// TIA Portal project "03PLC" (V15)

(* hardware
DEVICE "S7-1200 station_1"  S7-1200 Station
   slot 0: "Rack_0"  S7-1200 Rack  Rack  V1.0
   slot 1: "PLC_1"  CPU 1215C DC/DC/DC  6ES7 215-1AG40-0XB0  V4.0
   slot 2: "DI 16x24VDC/DQ 16xRelay_1"  SM 1223 DI16/DQ16 x relay  6ES7 223-1PL32-0XB0  V2.0
   slot 3: "DI 16x24VDC/DQ 16xRelay_2"  SM 1223 DI16/DQ16 x relay  6ES7 223-1PL32-0XB0  V2.0
   slot 4: "DI 16x24VDC_1"  6ES7 221-1BH32-0XB0  V2.0
   slot 5: "DI 16x24VDC_2"  6ES7 221-1BH32-0XB0  V2.0
DEVICE "HMI_1"  TP700 Comfort
   slot 0: "HMI_1"  TP700 Comfort  6AV2 124-0GC01-0AX0  15.0.0.0
   slot 1: "HMI_RT_1"  TP700 Comfort  6AV2 124-0GC01-0AX0  15.0.0.0
   slot 5: "HMI_1.IE_CP_1"  PROFINET Interface  15.0.0.0
      slot 1: "PROFINET Interface_1"  PROFINET Interface
         slot 1: "Port_1"  Port
         slot 2: "Port_2"  Port
   slot 7: "HMI_1.MPI/DP_CP_1"  MPI/DP Interface  15.0.0.0
DEVICE "GSD device_1"  GSD.Device.PN
   slot 0: "机架"  Rack  V1.0
   slot 0: "RFID"  RF180C V2.2  6GT2 002-0JD00  2.0
      slot 0: "Standard"  Standard
      slot 1: "RF180C Interface"  RF180C Interface
         slot 1: "Port 1"  Port 1
         slot 2: "Port 2"  Port 2
      slot 1: "2x RS422 channels RFID_1"  2x RS422 channels RFID
         slot 0: "2x RS422 channels RFID"  2x RS422 channels RFID
*)

// ===== PLC "PLC_1"  CPU 1215C DC/DC/DC =====

VAR_GLOBAL   // PLC tag table "默认变量表"
   "System_Byte" AT %MB1 : Byte;
   "FirstScan" AT %M1.0 : Bool;
   "DiagStatusUpdate" AT %M1.1 : Bool;
   "AlwaysTRUE" AT %M1.2 : Bool;
   "AlwaysFALSE" AT %M1.3 : Bool;
   "Clock_Byte" AT %MB0 : Byte;
   "Clock_10Hz" AT %M0.0 : Bool;
   "Clock_5Hz" AT %M0.1 : Bool;
   "Clock_2.5Hz" AT %M0.2 : Bool;
   "Clock_2Hz" AT %M0.3 : Bool;
   "Clock_1.25Hz" AT %M0.4 : Bool;
   "Clock_1Hz" AT %M0.5 : Bool;
   "Clock_0.625Hz" AT %M0.6 : Bool;
   "Clock_0.5Hz" AT %M0.7 : Bool;
   "Tag_1" AT %M9.0 : Bool;
   "Tag_2" AT %MW10 : Word;
   "Tag_69" AT %M100.0 : Bool;
   "Tag_70" AT %M200.0 : Bool;
   "Tag_71" AT %I0.2 : Bool;
   "Tag_72" AT %Q5.0 : Bool;
END_VAR

VAR_GLOBAL   // PLC tag table "变量表_1"
   "Tag_3" AT %I2.0 : Bool;
   "Tag_4" AT %I2.1 : Bool;
   "Tag_5" AT %I2.2 : Bool;
   "Tag_6" AT %I2.3 : Bool;
   "Tag_7" AT %I2.4 : Bool;
   "Tag_8" AT %I2.5 : Bool;
   "Tag_9" AT %I2.6 : Bool;
   "Tag_10" AT %I2.7 : Bool;
   "Tag_11" AT %Q2.0 : Bool;
   "Tag_12" AT %Q2.1 : Bool;
   "Tag_13" AT %Q2.2 : Bool;
   "Tag_14" AT %Q2.3 : Bool;
   "Tag_15" AT %Q2.4 : Bool;
   "Tag_16" AT %Q2.5 : Bool;
   "Tag_17" AT %Q2.6 : Bool;
   "Tag_18" AT %Q2.7 : Bool;
   "Tag_19" AT %I3.0 : Bool;
   "Tag_20" AT %I5.0 : Bool;
   "Tag_21" AT %I5.2 : Bool;
   "Tag_22" AT %Q0.4 : Bool;
   "Tag_23" AT %Q0.5 : Bool;
END_VAR

VAR_GLOBAL   // PLC tag table "变量表_2"
   "Tag_24" AT %I4.0 : Bool;
   "Tag_25" AT %I4.1 : Bool;
   "Tag_26" AT %I4.2 : Bool;
   "Tag_27" AT %I4.3 : Bool;
   "Tag_28" AT %I4.4 : Bool;
   "Tag_29" AT %I4.5 : Bool;
   "Tag_30" AT %I4.6 : Bool;
   "Tag_31" AT %Q4.0 : Bool;
   "Tag_32" AT %Q4.1 : Bool;
   "Tag_33" AT %Q4.2 : Bool;
   "Tag_34" AT %Q4.3 : Bool;
   "Tag_35" AT %Q4.4 : Bool;
   "Tag_36" AT %Q4.5 : Bool;
   "Tag_37" AT %Q4.6 : Bool;
   "Tag_38" AT %Q4.7 : Bool;
END_VAR

VAR_GLOBAL   // PLC tag table "变量表_3"
   "Tag_39" AT %I6.0 : Bool;
   "Tag_40" AT %I6.1 : Bool;
   "Tag_41" AT %I6.2 : Bool;
   "Tag_42" AT %I6.3 : Bool;
   "Tag_43" AT %I6.4 : Bool;
   "Tag_44" AT %I6.5 : Bool;
   "Tag_45" AT %I6.6 : Bool;
   "Tag_46" AT %I6.7 : Bool;
   "Tag_47" AT %I7.0 : Bool;
   "Tag_48" AT %I7.1 : Bool;
   "Tag_49" AT %I7.2 : Bool;
   "Tag_50" AT %I7.3 : Bool;
   "Tag_51" AT %I7.4 : Bool;
   "Tag_52" AT %I7.5 : Bool;
   "Tag_53" AT %I7.6 : Bool;
   "Tag_54" AT %I8.0 : Bool;
   "Tag_55" AT %I8.1 : Bool;
   "Tag_56" AT %I8.2 : Bool;
   "Tag_57" AT %I8.3 : Bool;
   "Tag_58" AT %I8.4 : Bool;
   "Tag_59" AT %I8.5 : Bool;
   "Tag_60" AT %I8.6 : Bool;
   "Tag_61" AT %I8.7 : Bool;
   "Tag_62" AT %I9.0 : Bool;
   "Tag_63" AT %I9.1 : Bool;
   "Tag_64" AT %I9.2 : Bool;
   "Tag_65" AT %I9.3 : Bool;
   "Tag_66" AT %I9.4 : Bool;
   "Tag_67" AT %I9.5 : Bool;
   "Tag_68" AT %I9.6 : Bool;
END_VAR

TYPE "用户数据类型_1"
   STRUCT
      场次 : Int;
      种类 : Int;
      材质 : Int;
      状态 : Int;
   END_STRUCT;
END_TYPE

DATA_BLOCK "mes数据块"   // DB1
{ S7_Optimized_Access := 'FALSE' }
VERSION : 0.1
   VAR
      mes给plc : Struct
         mes命令 : Struct
            "1" : Int;
            "2" : Int;
            "3" : Int;
            "4" : Int;
            "5" : Int;
            "6" : Int;
            "7" : Int;
            "8" : Int;
            "9" : Int;
            "10" : Int;
         END_STRUCT;
         mes反馈车床 : Struct
            "1" : Int;
            "2" : Int;
            "3" : Int;
            "4" : Int;
            "5" : Int;
         END_STRUCT;
         mes反馈cnc : Struct
            "1" : Int;
            "2" : Int;
            "3" : Int;
            "4" : Int;
            "5" : Int;
         END_STRUCT;
      END_STRUCT;
      plc给mes : Struct
         plc命令车床 : Struct
            "1" : Int;
            "2" : Int;
            "3" : Int;
            "4" : Int;
            "5" : Int;
         END_STRUCT;
         plc命令cnc : Struct
            "1" : Int;
            "2" : Int;
            "3" : Int;
            "4" : Int;
            "5" : Int;
         END_STRUCT;
         plc反馈 : Struct
            "1" : Int;
            "2" : Int;
            "3" : Int;
            "4" : Int;
            "5" : Int;
            "6" : Int;
            "7" : Int;
            "8" : Int;
            "9" : Int;
            "10" : Int;
         END_STRUCT;
         机器人状态 : Struct
            "1" : Int;
            "2" : Int;
            "3" : Int;
            "4" : Int;
            "5" : Int;
            "6" : Int;
            "7" : Int;
            "8" : Int;
            "9" : Int;
            "10" : Int;
            "11" : Int;
         END_STRUCT;
         保留 : Array[0..8] of Word;
      END_STRUCT;
      仓库 : Struct
         "1" : Bool;
         "2" : Bool;
         "3" : Bool;
         "4" : Bool;
         "5" : Bool;
         "6" : Bool;
         "7" : Bool;
         "8" : Bool;
         "9" : Bool;
         "10" : Bool;
         "11" : Bool;
         "12" : Bool;
         "13" : Bool;
         "14" : Bool;
         "15" : Bool;
         保留 : Bool;
         "16" : Bool;
         "17" : Bool;
         "18" : Bool;
         "19" : Bool;
         "20" : Bool;
         "21" : Bool;
         "22" : Bool;
         "23" : Bool;
         "24" : Bool;
         "25" : Bool;
         "26" : Bool;
         "27" : Bool;
         "28" : Bool;
         "29" : Bool;
         "30" : Bool;
      END_STRUCT;
      保留 : Array[0..47] of Bool;
      机床状态 : Array[0..79] of Bool;
      工件 : Array[1..30] of "用户数据类型_1";
      测量 : Array[1..10] of Int;
   END_VAR
BEGIN
END_DATA_BLOCK

DATA_BLOCK "机器人数据块"   // DB2
{ S7_Optimized_Access := 'FALSE' }
VERSION : 0.1
   VAR
      plc给机器人 : Struct
         "1" : Int;
         "2" : Int;
         "3" : Int;
         "4" : Int;
         "5" : Int;
         "6" : Int;
         "7" : Int;
         "8" : Int;
         "9" : Int;
         "10" : Int;
         "11" : Int;
         "12" : Int;
         "13" : Int;
         "14" : Int;
         "15" : Int;
         "16" : Int;
      END_STRUCT;
      机器人给plc : Struct
         "1" : Int;
         "2" : Int;
         "3" : Int;
         "4" : Int;
         "5" : Int;
         "6" : Int;
         "7" : Int;
         "8" : Int;
         "9" : Int;
         "10" : Int;
         "11" : Int;
         "12" : Int;
         "13" : Int;
         "14" : Int;
         "15" : Int;
         "16" : Int;
      END_STRUCT;
      机器人状态 : Struct
         "1" : Real;
         "2" : Real;
         "3" : Real;
         "4" : Real;
         "5" : Real;
         "6" : Real;
         "7" : Real;
         "8" : Real;
         "9" : Real;
         "10" : Real;
         "11" : Real;
         "12" : Real;
         "13" : Real;
         "14" : Real;
         "15" : Real;
         "16" : Real;
      END_STRUCT;
   END_VAR
BEGIN
END_DATA_BLOCK

DATA_BLOCK "hmi"   // DB3
{ S7_Optimized_Access := 'TRUE' }
VERSION : 0.1
   VAR
      车床卡盘 : Bool;
      cnc卡盘 : Bool;
      零点夹具 : Bool;
      车床门开关 : Bool;
      铣床门开关 : Bool;
      机器人home位 : Bool;
      mes订单已下发 : Bool;
      自动 : Bool;
      手动 : Bool;
      清理 : Time;
      间隔 : Time;
      种类 : Int;
      状态 : Int;
      当前仓位 : Int;
   END_VAR
BEGIN
END_DATA_BLOCK

DATA_BLOCK "mes_DB"   // DB4
{ S7_Optimized_Access := 'TRUE' }
VERSION : 0.1
// stored: InstanceOfName mes
"mes"
BEGIN
END_DATA_BLOCK

DATA_BLOCK "rfid_DB"   // DB7
{ S7_Optimized_Access := 'TRUE' }
VERSION : 0.1
// stored: InstanceOfName rfid
"rfid"
BEGIN
END_DATA_BLOCK

DATA_BLOCK "车床_DB"   // DB8
{ S7_Optimized_Access := 'TRUE' }
VERSION : 0.1
// stored: InstanceOfName 车床
"车床"
BEGIN
END_DATA_BLOCK

DATA_BLOCK "铣床_DB"   // DB9
{ S7_Optimized_Access := 'TRUE' }
VERSION : 0.1
// stored: InstanceOfName 铣床
"铣床"
BEGIN
END_DATA_BLOCK

DATA_BLOCK "机器人通讯_DB"   // DB10
{ S7_Optimized_Access := 'TRUE' }
VERSION : 0.1
// stored: InstanceOfName 机器人通讯
"机器人通讯"
BEGIN
END_DATA_BLOCK

DATA_BLOCK "机床状态_DB"   // DB11
{ S7_Optimized_Access := 'TRUE' }
VERSION : 0.1
// stored: InstanceOfName 机床状态
"机床状态"
BEGIN
END_DATA_BLOCK

DATA_BLOCK "测量_DB"   // DB12
{ S7_Optimized_Access := 'TRUE' }
VERSION : 0.1
// stored: InstanceOfName 测量
"测量"
BEGIN
END_DATA_BLOCK

DATA_BLOCK "有无料_DB"   // DB13
{ S7_Optimized_Access := 'TRUE' }
VERSION : 0.1
// stored: InstanceOfName 有无料
"有无料"
BEGIN
END_DATA_BLOCK

// folder: rfid

DATA_BLOCK "connect"   // DB5
{ S7_Optimized_Access := 'TRUE' }
VERSION : 0.1
   VAR
      connect : IID_HW_CONNECT;
   END_VAR
BEGIN
END_DATA_BLOCK

DATA_BLOCK "读写"   // DB6
{ S7_Optimized_Access := 'FALSE' }
VERSION : 0.1
   VAR
      读 : Array[0..1024] of Byte;
      写 : Array[0..1024] of Byte;
   END_VAR
BEGIN
END_DATA_BLOCK

// folder: (top level)

FUNCTION_BLOCK "机器人通讯"   // FB1, LAD
{ S7_Optimized_Access := 'TRUE' }
VERSION : 0.1
   VAR
      MB_CLIENT_Instance : MB_CLIENT;
      w1 : Bool;
      w2 : Bool;
      w3 : Bool;
      m1 : Bool;
      m2 : Bool;
      m3 : Bool;
      c1 : Bool;
      c2 : Bool;
      c3 : Bool;
      s1 : Word;
      s2 : Word;
      s3 : Word;
      轴1 : Int;
      轴2 : Int;
      轴3 : Int;
      轴4 : Int;
      轴5 : Int;
      轴6 : Int;
      轴7 : Int;
   END_VAR
BEGIN

REGION Network 1
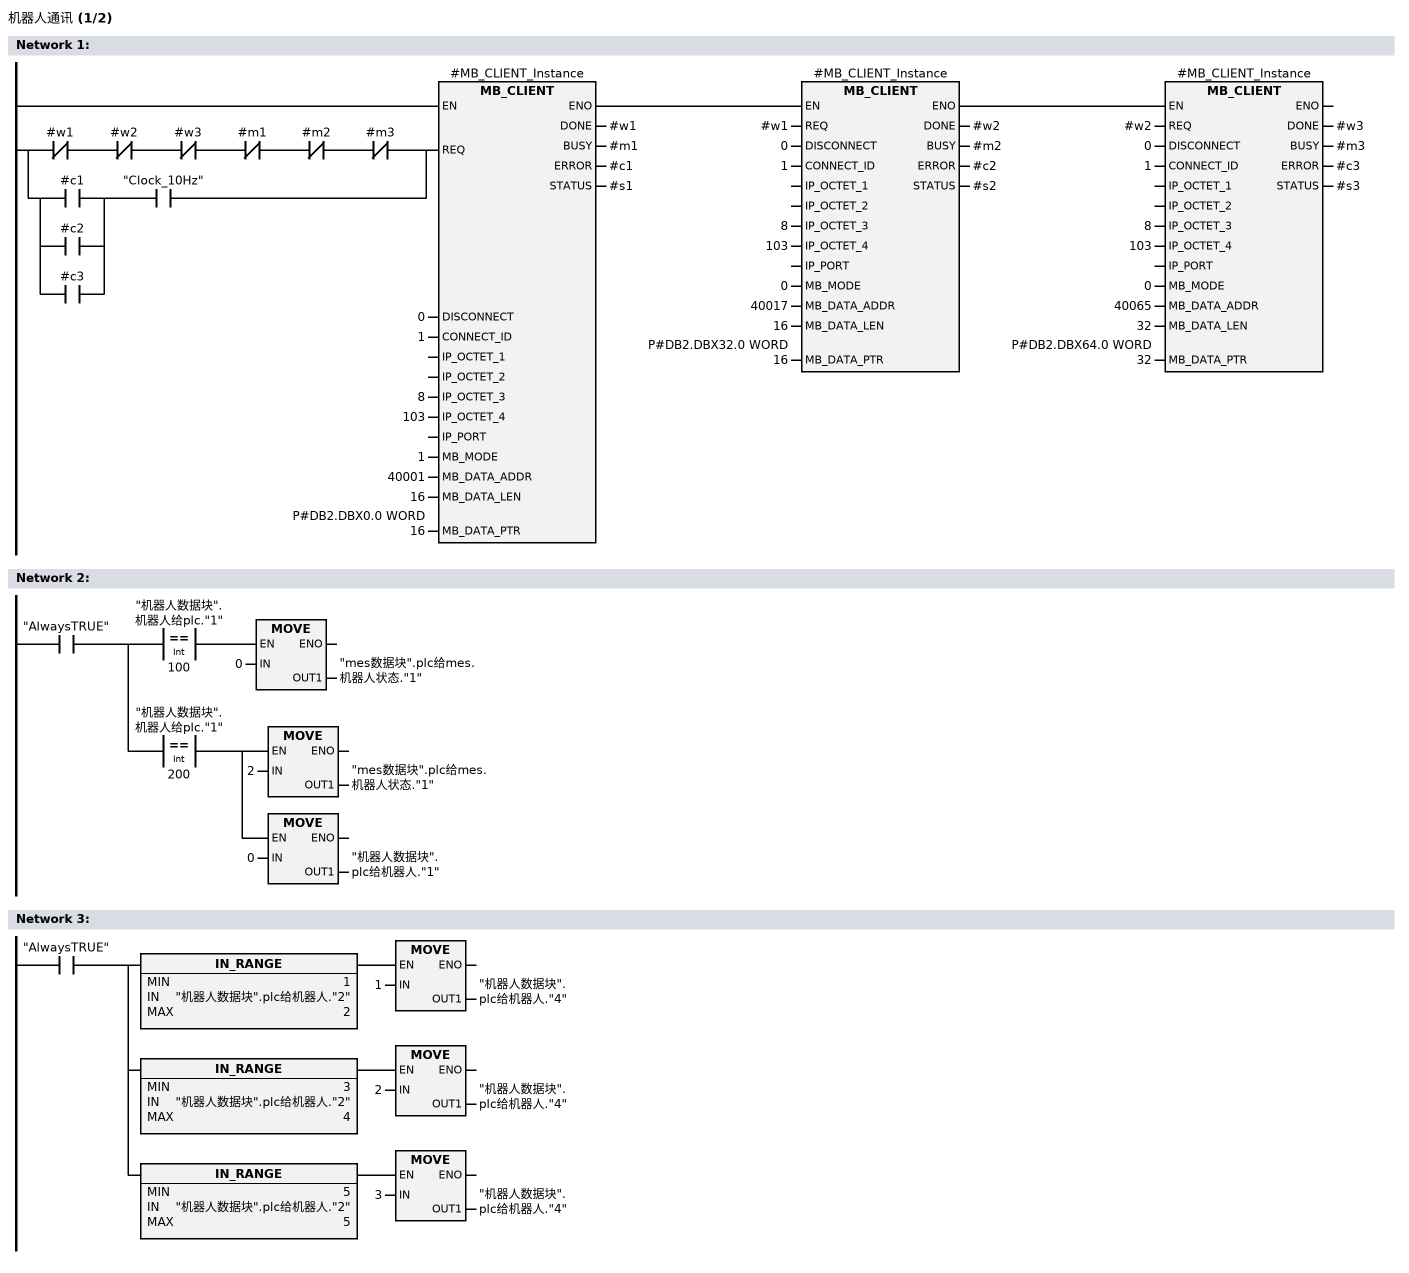
   // ENO of a box is taken as its EN; it also drops when the box reports an error
   #MB_CLIENT_Instance(REQ := (NOT #w1 AND NOT #w2 AND NOT #w3 AND NOT #m1 AND NOT #m2 AND NOT #m3) OR ((#c1 OR #c2 OR #c3) AND "Clock_10Hz"),   // MB_CLIENT
                       DISCONNECT := 0,
                       CONNECT_ID := 1,
                       IP_OCTET_3 := 8,
                       IP_OCTET_4 := 103,
                       MB_MODE := 1,
                       MB_DATA_ADDR := 40001,
                       MB_DATA_LEN := 16,
                       MB_DATA_PTR := P#DB2.DBX0.0 WORD 16,
                       DONE => #w1,
                       BUSY => #m1,
                       ERROR => #c1,
                       STATUS => #s1);
   #MB_CLIENT_Instance(REQ := #w1,   // MB_CLIENT
                       DISCONNECT := 0,
                       CONNECT_ID := 1,
                       IP_OCTET_3 := 8,
                       IP_OCTET_4 := 103,
                       MB_MODE := 0,
                       MB_DATA_ADDR := 40017,
                       MB_DATA_LEN := 16,
                       MB_DATA_PTR := P#DB2.DBX32.0 WORD 16,
                       DONE => #w2,
                       BUSY => #m2,
                       ERROR => #c2,
                       STATUS => #s2);
   #MB_CLIENT_Instance(REQ := #w2,   // MB_CLIENT
                       DISCONNECT := 0,
                       CONNECT_ID := 1,
                       IP_OCTET_3 := 8,
                       IP_OCTET_4 := 103,
                       MB_MODE := 0,
                       MB_DATA_ADDR := 40065,
                       MB_DATA_LEN := 32,
                       MB_DATA_PTR := P#DB2.DBX64.0 WORD 32,
                       DONE => #w3,
                       BUSY => #m3,
                       ERROR => #c3,
                       STATUS => #s3);
END_REGION

REGION Network 2
   RUNG wire#powerrail
      Contact( "AlwaysTRUE" )
      wire#w1
      { S7_Templates := "SrcType := Int" } EQ_Contact(in1 := "机器人数据块".机器人给plc."1", in2 := 100)
      Move(in := 0, out1 => "mes数据块".plc给mes.机器人状态."1")
   END_RUNG
   RUNG wire#w1
      { S7_Templates := "SrcType := Int" } EQ_Contact(in1 := "机器人数据块".机器人给plc."1", in2 := 200)
      wire#w2
      Move(in := 2, out1 => "mes数据块".plc给mes.机器人状态."1")
   END_RUNG
   RUNG wire#w2
      Move(in := 0, out1 => "机器人数据块".plc给机器人."1")
   END_RUNG
   // the same network as SCL:
   IF "AlwaysTRUE" AND ("机器人数据块".机器人给plc."1" = 100) THEN "mes数据块".plc给mes.机器人状态."1" := 0; END_IF;
   IF "AlwaysTRUE" AND ("机器人数据块".机器人给plc."1" = 200) THEN
       "mes数据块".plc给mes.机器人状态."1" := 2;
       "机器人数据块".plc给机器人."1" := 0;
   END_IF;
END_REGION

REGION Network 3
   RUNG wire#powerrail
      Contact( "AlwaysTRUE" )
      wire#w1
      { S7_Templates := "SrcType := Int" } InRange(min := 1, in := "机器人数据块".plc给机器人."2", max := 2)
      Move(in := 1, out1 => "机器人数据块".plc给机器人."4")
   END_RUNG
   RUNG wire#w1
      { S7_Templates := "SrcType := Int" } InRange(min := 3, in := "机器人数据块".plc给机器人."2", max := 4)
      Move(in := 2, out1 => "机器人数据块".plc给机器人."4")
   END_RUNG
   RUNG wire#w1
      { S7_Templates := "SrcType := Int" } InRange(min := 5, in := "机器人数据块".plc给机器人."2", max := 5)
      Move(in := 3, out1 => "机器人数据块".plc给机器人."4")
   END_RUNG
   // the same network as SCL:
   IF "AlwaysTRUE" AND (1 <= "机器人数据块".plc给机器人."2") AND ("机器人数据块".plc给机器人."2" <= 2) THEN
       "机器人数据块".plc给机器人."4" := 1;
   END_IF;
   IF "AlwaysTRUE" AND (3 <= "机器人数据块".plc给机器人."2") AND ("机器人数据块".plc给机器人."2" <= 4) THEN
       "机器人数据块".plc给机器人."4" := 2;
   END_IF;
   IF "AlwaysTRUE" AND (5 <= "机器人数据块".plc给机器人."2") AND ("机器人数据块".plc给机器人."2" <= 5) THEN
       "机器人数据块".plc给机器人."4" := 3;
   END_IF;
END_REGION

REGION Network 4
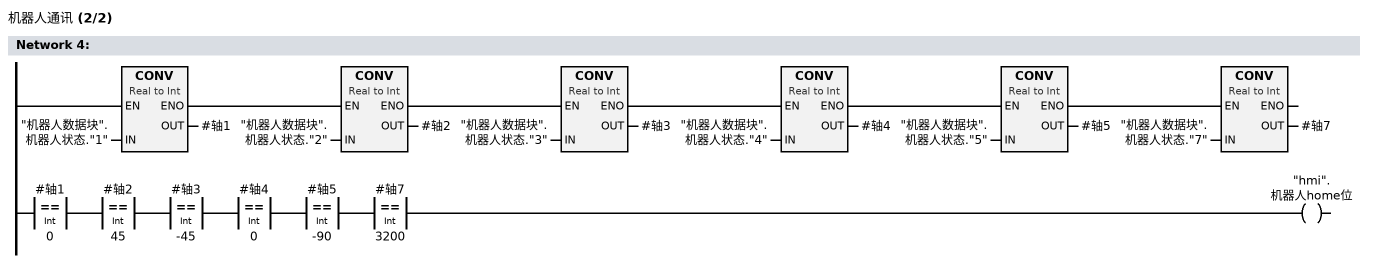
   RUNG wire#powerrail
      { S7_Templates := "[SrcType := Real, DestType := Int]" } Convert(in := "机器人数据块".机器人状态."1", out => #轴1)
      { S7_Templates := "[SrcType := Real, DestType := Int]" } Convert(in := "机器人数据块".机器人状态."2", out => #轴2)
      { S7_Templates := "[SrcType := Real, DestType := Int]" } Convert(in := "机器人数据块".机器人状态."3", out => #轴3)
      { S7_Templates := "[SrcType := Real, DestType := Int]" } Convert(in := "机器人数据块".机器人状态."4", out => #轴4)
      { S7_Templates := "[SrcType := Real, DestType := Int]" } Convert(in := "机器人数据块".机器人状态."5", out => #轴5)
      { S7_Templates := "[SrcType := Real, DestType := Int]" } Convert(in := "机器人数据块".机器人状态."7", out => #轴7)
   END_RUNG
   RUNG wire#powerrail
      { S7_Templates := "SrcType := Int" } EQ_Contact(in1 := #轴1, in2 := 0)
      { S7_Templates := "SrcType := Int" } EQ_Contact(in1 := #轴2, in2 := 45)
      { S7_Templates := "SrcType := Int" } EQ_Contact(in1 := #轴3, in2 := -45)
      { S7_Templates := "SrcType := Int" } EQ_Contact(in1 := #轴4, in2 := 0)
      { S7_Templates := "SrcType := Int" } EQ_Contact(in1 := #轴5, in2 := -90)
      { S7_Templates := "SrcType := Int" } EQ_Contact(in1 := #轴7, in2 := 3200)
      Coil( "hmi".机器人home位 )
   END_RUNG
   // the same network as SCL:
   #轴1 := REAL_TO_INT("机器人数据块".机器人状态."1");
   #轴2 := REAL_TO_INT("机器人数据块".机器人状态."2");
   #轴3 := REAL_TO_INT("机器人数据块".机器人状态."3");
   #轴4 := REAL_TO_INT("机器人数据块".机器人状态."4");
   #轴5 := REAL_TO_INT("机器人数据块".机器人状态."5");
   #轴7 := REAL_TO_INT("机器人数据块".机器人状态."7");
   "hmi".机器人home位 := (#轴1 = 0) AND (#轴2 = 45) AND (#轴3 = (-45)) AND (#轴4 = 0) AND (#轴5 = (-90)) AND (#轴7 = 3200);
END_REGION
END_FUNCTION_BLOCK

FUNCTION "位置" : Void   // FC1, SCL
{ S7_Optimized_Access := 'TRUE' }
VERSION : 0.1
   VAR_INPUT
      取 : Int;
      放 : Int;
   END_VAR
   VAR_OUTPUT
      行 : Int;
      列 : Int;
      当前仓位 : Int;
      种类 : Int;
      状态 : Int;
   END_VAR
BEGIN
   #当前仓位 := #取 + #放;
   #行 := (#当前仓位 - 1) / 6 + 1;
   #列 := (#当前仓位 - 1) MOD 6 + 1;
   IF #当前仓位>0 THEN
       #种类 := "mes数据块".工件[#当前仓位].种类;
       #状态 := "mes数据块".工件[#当前仓位].状态;
           // Statement section IF
       ;
   END_IF;
END_FUNCTION

ORGANIZATION_BLOCK "Main"   // OB1, LAD, ProgramCycle
TITLE = "Main Program Sweep (Cycle)"
{ S7_Optimized_Access := 'TRUE' }
VERSION : 0.1
   VAR_INPUT
      Initial_Call : Bool;   // Initial call of this OB
      Remanence : Bool;   // =True, if remanent data are available
   END_VAR
   VAR_TEMP   // added for the SCL form of the ladder/FBD networks
      _w1 : Bool;
      _w2 : Bool;
      _w3 : Bool;
   END_VAR
BEGIN

REGION Network 1
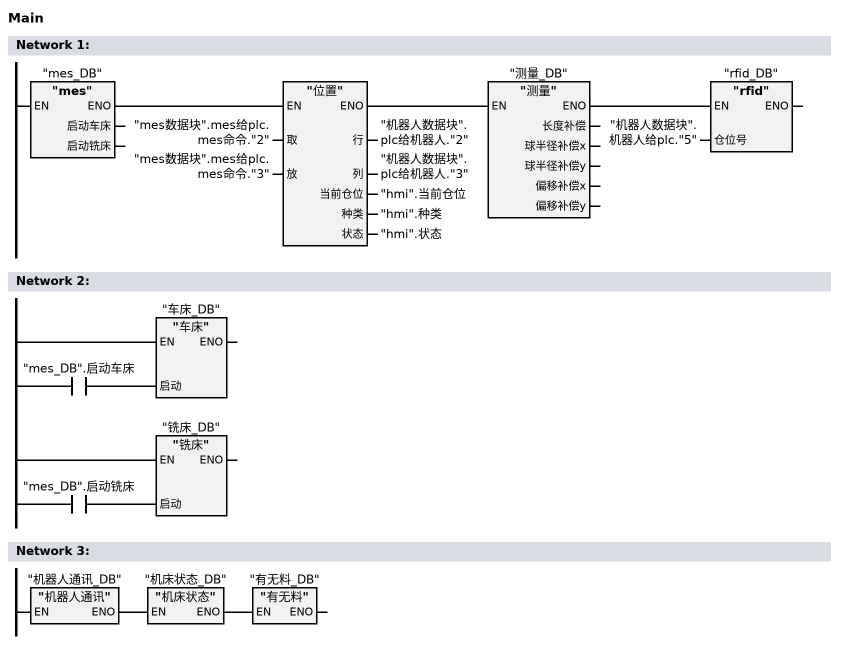
   RUNG wire#powerrail
      "mes_DB"(启动车床 =>, 启动铣床 =>)
      "位置"(取 := "mes数据块".mes给plc.mes命令."2", 放 := "mes数据块".mes给plc.mes命令."3", 行 => "机器人数据块".plc给机器人."2", 列 => "机器人数据块".plc给机器人."3", 当前仓位 => "hmi".当前仓位, 种类 => "hmi".种类, 状态 => "hmi".状态)
      "测量_DB"(长度补偿 =>, 球半径补偿x =>, 球半径补偿y =>, 偏移补偿x =>, 偏移补偿y =>)
      "rfid_DB"(仓位号 := "机器人数据块".机器人给plc."5")
   END_RUNG
   // the same network as SCL:
   "mes_DB"(ENO => #_w1);   // "mes"
   "位置"(EN := #_w1,
        取 := "mes数据块".mes给plc.mes命令."2",
        放 := "mes数据块".mes给plc.mes命令."3",
        行 => "机器人数据块".plc给机器人."2",
        列 => "机器人数据块".plc给机器人."3",
        当前仓位 => "hmi".当前仓位,
        种类 => "hmi".种类,
        状态 => "hmi".状态,
        ENO => #_w2);
   "测量_DB"(EN := #_w2, ENO => #_w3);   // "测量"
   IF #_w3 THEN
       "rfid_DB"(仓位号 := "机器人数据块".机器人给plc."5");   // "rfid"
   END_IF;
END_REGION

REGION Network 2
   RUNG wire#powerrail
      "车床_DB"(启动 := wire#w1)
   END_RUNG
   RUNG wire#powerrail
      Contact( "mes_DB".启动车床 )
   END_RUNG wire#w1
   RUNG wire#powerrail
      "铣床_DB"(启动 := wire#w2)
   END_RUNG
   RUNG wire#powerrail
      Contact( "mes_DB".启动铣床 )
   END_RUNG wire#w2
   // the same network as SCL:
   "车床_DB"(启动 := "mes_DB".启动车床);   // "车床"
   "铣床_DB"(启动 := "mes_DB".启动铣床);   // "铣床"
END_REGION

REGION Network 3
   RUNG wire#powerrail
      "机器人通讯_DB"()
      "机床状态_DB"()
      "有无料_DB"()
   END_RUNG
   // the same network as SCL:
   "机器人通讯_DB"(ENO => #_w1);   // "机器人通讯"
   "机床状态_DB"(EN := #_w1, ENO => #_w2);   // "机床状态"
   IF #_w2 THEN
       "有无料_DB"();   // "有无料"
   END_IF;
END_REGION
END_ORGANIZATION_BLOCK

// folder: mes

FUNCTION_BLOCK "plc解析"   // FB2, LAD
{ S7_Optimized_Access := 'TRUE' }
VERSION : 0.1
   VAR_INPUT
      启动 : Bool;
      mes反馈 : Int;
      命令码 : Int;
   END_VAR
   VAR_OUTPUT
      完成 : Bool;
   END_VAR
   VAR_IN_OUT
      plc命令 : Int;
   END_VAR
   VAR
      "step" : Word;
   END_VAR
   VAR_TEMP   // added for the SCL form of the ladder/FBD networks
      _w1 : Bool;
   END_VAR
BEGIN

REGION Network 1
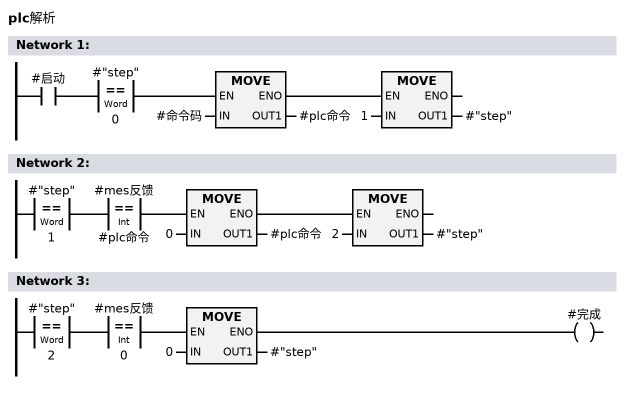
   RUNG wire#powerrail
      Contact( #启动 )
      { S7_Templates := "SrcType := Word" } EQ_Contact(in1 := #"step", in2 := 0)
      Move(in := #命令码, out1 => #plc命令)
      Move(in := 1, out1 => #"step")
   END_RUNG
   // the same network as SCL:
   IF #启动 AND (#"step" = 0) THEN
       #plc命令 := #命令码;
       #"step" := 1;
   END_IF;
END_REGION

REGION Network 2
   RUNG wire#powerrail
      { S7_Templates := "SrcType := Word" } EQ_Contact(in1 := #"step", in2 := 1)
      { S7_Templates := "SrcType := Int" } EQ_Contact(in1 := #mes反馈, in2 := #plc命令)
      Move(in := 0, out1 => #plc命令)
      Move(in := 2, out1 => #"step")
   END_RUNG
   // the same network as SCL:
   #_w1 := (#"step" = 1) AND (#mes反馈 = #plc命令);
   IF #_w1 THEN
       #plc命令 := 0;
       #"step" := 2;
   END_IF;
END_REGION

REGION Network 3
   RUNG wire#powerrail
      { S7_Templates := "SrcType := Word" } EQ_Contact(in1 := #"step", in2 := 2)
      { S7_Templates := "SrcType := Int" } EQ_Contact(in1 := #mes反馈, in2 := 0)
      Move(in := 0, out1 => #"step")
      Coil( #完成 )
   END_RUNG
   // the same network as SCL:
   #_w1 := (#"step" = 2) AND (#mes反馈 = 0);
   IF #_w1 THEN #"step" := 0; END_IF;
   #完成 := #_w1;
END_REGION
END_FUNCTION_BLOCK

FUNCTION_BLOCK "mes解析"   // FB3, LAD
{ S7_Optimized_Access := 'TRUE' }
VERSION : 0.1
   VAR_INPUT
      命令码 : Int;
      mes命令 : Int;
   END_VAR
   VAR_OUTPUT
      完成 : Bool;
   END_VAR
   VAR_IN_OUT
      plc反馈 : Int;
   END_VAR
   VAR
      "step" : Word;
   END_VAR
   VAR_TEMP   // added for the SCL form of the ladder/FBD networks
      _w1 : Bool;
   END_VAR
BEGIN

REGION Network 1
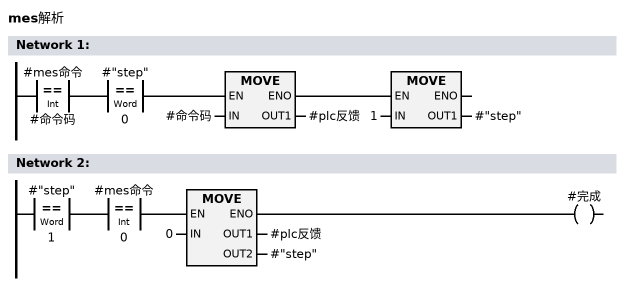
   RUNG wire#powerrail
      { S7_Templates := "SrcType := Int" } EQ_Contact(in1 := #mes命令, in2 := #命令码)
      { S7_Templates := "SrcType := Word" } EQ_Contact(in1 := #"step", in2 := 0)
      Move(in := #命令码, out1 => #plc反馈)
      Move(in := 1, out1 => #"step")
   END_RUNG
   // the same network as SCL:
   IF (#mes命令 = #命令码) AND (#"step" = 0) THEN
       #plc反馈 := #命令码;
       #"step" := 1;
   END_IF;
END_REGION

REGION Network 2
   RUNG wire#powerrail
      { S7_Templates := "SrcType := Word" } EQ_Contact(in1 := #"step", in2 := 1)
      { S7_Templates := "SrcType := Int" } EQ_Contact(in1 := #mes命令, in2 := 0)
      Move(in := 0, out1 => #plc反馈, out2 => #"step")
      Coil( #完成 )
   END_RUNG
   // the same network as SCL:
   #_w1 := (#"step" = 1) AND (#mes命令 = 0);
   IF #_w1 THEN
       #plc反馈 := 0;
       #"step" := 0;
   END_IF;
   #完成 := #_w1;
END_REGION
END_FUNCTION_BLOCK

FUNCTION_BLOCK "mes"   // FB4, LAD
{ S7_Optimized_Access := 'TRUE' }
VERSION : 0.1
   VAR_OUTPUT
      启动车床 : Bool;
      启动铣床 : Bool;
   END_VAR
   VAR
      车床程序 : Bool;
      铣床程序 : Bool;
      MB_SERVER_Instance : MB_SERVER;
      mes解析_Instance : "mes解析";
      mes解析_Instance_1 : "mes解析";
      mes解析_Instance_2 : "mes解析";
      mes解析_Instance_3 : "mes解析";
      plc解析_Instance : "plc解析";
      plc解析_Instance_1 : "plc解析";
      IEC_Timer_0_Instance : TON_TIME;
      IEC_Timer_0_Instance_1 : TON_TIME;
   END_VAR
   VAR_TEMP   // added for the SCL form of the ladder/FBD networks
      _w1 : Bool;
      _w2 : Bool;
      _w3 : Bool;
      _w4 : Bool;
      _w5 : Bool;
      _w6 : Bool;
   END_VAR
BEGIN

REGION Network 1
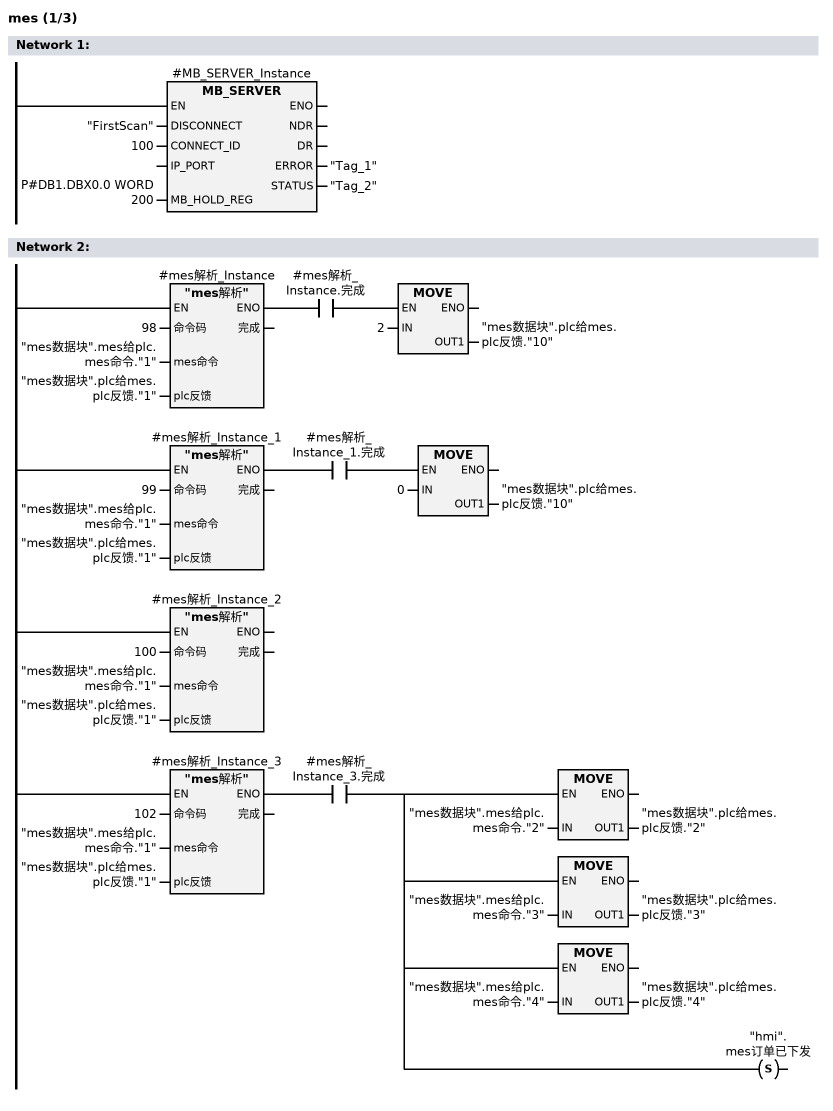
   #MB_SERVER_Instance(DISCONNECT := "FirstScan",   // MB_SERVER
                       CONNECT_ID := 100,
                       MB_HOLD_REG := P#DB1.DBX0.0 WORD 200,
                       ERROR => "Tag_1",
                       STATUS => "Tag_2");
END_REGION

REGION Network 2
   RUNG wire#powerrail
      #mes解析_Instance(命令码 := 98, mes命令 := "mes数据块".mes给plc.mes命令."1", plc反馈 := "mes数据块".plc给mes.plc反馈."1", 完成 =>)
      Contact( #mes解析_Instance.完成 )
      Move(in := 2, out1 => "mes数据块".plc给mes.plc反馈."10")
   END_RUNG
   RUNG wire#powerrail
      #mes解析_Instance_1(命令码 := 99, mes命令 := "mes数据块".mes给plc.mes命令."1", plc反馈 := "mes数据块".plc给mes.plc反馈."1", 完成 =>)
      Contact( #mes解析_Instance_1.完成 )
      Move(in := 0, out1 => "mes数据块".plc给mes.plc反馈."10")
   END_RUNG
   RUNG wire#powerrail
      #mes解析_Instance_2(命令码 := 100, mes命令 := "mes数据块".mes给plc.mes命令."1", plc反馈 := "mes数据块".plc给mes.plc反馈."1", 完成 =>)
   END_RUNG
   RUNG wire#powerrail
      #mes解析_Instance_3(命令码 := 102, mes命令 := "mes数据块".mes给plc.mes命令."1", plc反馈 := "mes数据块".plc给mes.plc反馈."1", 完成 =>)
      Contact( #mes解析_Instance_3.完成 )
      wire#w1
      Move(in := "mes数据块".mes给plc.mes命令."2", out1 => "mes数据块".plc给mes.plc反馈."2")
   END_RUNG
   RUNG wire#w1
      Move(in := "mes数据块".mes给plc.mes命令."3", out1 => "mes数据块".plc给mes.plc反馈."3")
   END_RUNG
   RUNG wire#w1
      Move(in := "mes数据块".mes给plc.mes命令."4", out1 => "mes数据块".plc给mes.plc反馈."4")
   END_RUNG
   RUNG wire#w1
      S_Coil( "hmi".mes订单已下发 )
   END_RUNG
   // the same network as SCL:
   #mes解析_Instance(命令码 := 98,   // "mes解析"
                   mes命令 := "mes数据块".mes给plc.mes命令."1",
                   plc反馈 := "mes数据块".plc给mes.plc反馈."1",
                   ENO => #_w1);
   IF #_w1 AND #mes解析_Instance.完成 THEN "mes数据块".plc给mes.plc反馈."10" := 2; END_IF;
   #mes解析_Instance_1(命令码 := 99,   // "mes解析"
                     mes命令 := "mes数据块".mes给plc.mes命令."1",
                     plc反馈 := "mes数据块".plc给mes.plc反馈."1",
                     ENO => #_w2);
   IF #_w2 AND #mes解析_Instance_1.完成 THEN "mes数据块".plc给mes.plc反馈."10" := 0; END_IF;
   #mes解析_Instance_2(命令码 := 100, mes命令 := "mes数据块".mes给plc.mes命令."1", plc反馈 := "mes数据块".plc给mes.plc反馈."1");   // "mes解析"
   #mes解析_Instance_3(命令码 := 102,   // "mes解析"
                     mes命令 := "mes数据块".mes给plc.mes命令."1",
                     plc反馈 := "mes数据块".plc给mes.plc反馈."1",
                     ENO => #_w3);
   IF #_w3 AND #mes解析_Instance_3.完成 THEN
       "mes数据块".plc给mes.plc反馈."2" := "mes数据块".mes给plc.mes命令."2";
       "mes数据块".plc给mes.plc反馈."3" := "mes数据块".mes给plc.mes命令."3";
       "mes数据块".plc给mes.plc反馈."4" := "mes数据块".mes给plc.mes命令."4";
       "hmi".mes订单已下发 := TRUE;
   END_IF;
END_REGION

REGION Network 3
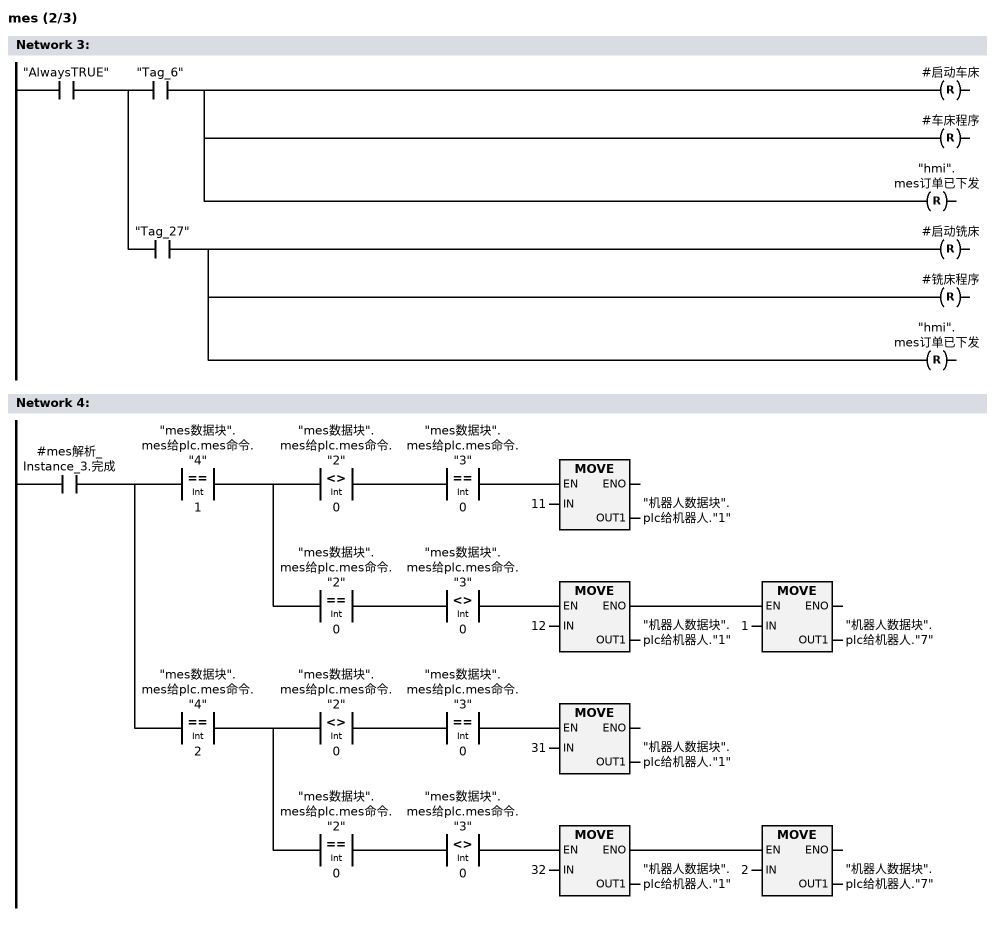
   RUNG wire#powerrail
      Contact( "AlwaysTRUE" )
      wire#w1
      Contact( "Tag_6" )
      wire#w2
      R_Coil( #启动车床 )
   END_RUNG
   RUNG wire#w2
      R_Coil( #车床程序 )
   END_RUNG
   RUNG wire#w2
      R_Coil( "hmi".mes订单已下发 )
   END_RUNG
   RUNG wire#w1
      Contact( "Tag_27" )
      wire#w3
      R_Coil( #启动铣床 )
   END_RUNG
   RUNG wire#w3
      R_Coil( #铣床程序 )
   END_RUNG
   RUNG wire#w3
      R_Coil( "hmi".mes订单已下发 )
   END_RUNG
   // the same network as SCL:
   IF "AlwaysTRUE" AND "Tag_6" THEN
       #启动车床 := FALSE;
       #车床程序 := FALSE;
       "hmi".mes订单已下发 := FALSE;
   END_IF;
   IF "AlwaysTRUE" AND "Tag_27" THEN
       #启动铣床 := FALSE;
       #铣床程序 := FALSE;
       "hmi".mes订单已下发 := FALSE;
   END_IF;
END_REGION

REGION Network 4
   RUNG wire#powerrail
      Contact( #mes解析_Instance_3.完成 )
      wire#w1
      { S7_Templates := "SrcType := Int" } EQ_Contact(in1 := "mes数据块".mes给plc.mes命令."4", in2 := 1)
      wire#w2
      { S7_Templates := "SrcType := Int" } NE_Contact(in1 := "mes数据块".mes给plc.mes命令."2", in2 := 0)
      { S7_Templates := "SrcType := Int" } EQ_Contact(in1 := "mes数据块".mes给plc.mes命令."3", in2 := 0)
      Move(in := 11, out1 => "机器人数据块".plc给机器人."1")
   END_RUNG
   RUNG wire#w2
      { S7_Templates := "SrcType := Int" } EQ_Contact(in1 := "mes数据块".mes给plc.mes命令."2", in2 := 0)
      { S7_Templates := "SrcType := Int" } NE_Contact(in1 := "mes数据块".mes给plc.mes命令."3", in2 := 0)
      Move(in := 12, out1 => "机器人数据块".plc给机器人."1")
      Move(in := 1, out1 => "机器人数据块".plc给机器人."7")
   END_RUNG
   RUNG wire#w1
      { S7_Templates := "SrcType := Int" } EQ_Contact(in1 := "mes数据块".mes给plc.mes命令."4", in2 := 2)
      wire#w3
      { S7_Templates := "SrcType := Int" } NE_Contact(in1 := "mes数据块".mes给plc.mes命令."2", in2 := 0)
      { S7_Templates := "SrcType := Int" } EQ_Contact(in1 := "mes数据块".mes给plc.mes命令."3", in2 := 0)
      Move(in := 31, out1 => "机器人数据块".plc给机器人."1")
   END_RUNG
   RUNG wire#w3
      { S7_Templates := "SrcType := Int" } EQ_Contact(in1 := "mes数据块".mes给plc.mes命令."2", in2 := 0)
      { S7_Templates := "SrcType := Int" } NE_Contact(in1 := "mes数据块".mes给plc.mes命令."3", in2 := 0)
      Move(in := 32, out1 => "机器人数据块".plc给机器人."1")
      Move(in := 2, out1 => "机器人数据块".plc给机器人."7")
   END_RUNG
   // the same network as SCL:
   #_w1 := #mes解析_Instance_3.完成 AND ("mes数据块".mes给plc.mes命令."4" = 1);
   IF #_w1 AND ("mes数据块".mes给plc.mes命令."2" <> 0) AND ("mes数据块".mes给plc.mes命令."3" = 0) THEN
       "机器人数据块".plc给机器人."1" := 11;
   END_IF;
   IF #_w1 AND ("mes数据块".mes给plc.mes命令."2" = 0) AND ("mes数据块".mes给plc.mes命令."3" <> 0) THEN
       "机器人数据块".plc给机器人."1" := 12;
       "机器人数据块".plc给机器人."7" := 1;
   END_IF;
   #_w2 := #mes解析_Instance_3.完成 AND ("mes数据块".mes给plc.mes命令."4" = 2);
   IF #_w2 AND ("mes数据块".mes给plc.mes命令."2" <> 0) AND ("mes数据块".mes给plc.mes命令."3" = 0) THEN
       "机器人数据块".plc给机器人."1" := 31;
   END_IF;
   IF #_w2 AND ("mes数据块".mes给plc.mes命令."2" = 0) AND ("mes数据块".mes给plc.mes命令."3" <> 0) THEN
       "机器人数据块".plc给机器人."1" := 32;
       "机器人数据块".plc给机器人."7" := 2;
   END_IF;
END_REGION

REGION Network 5
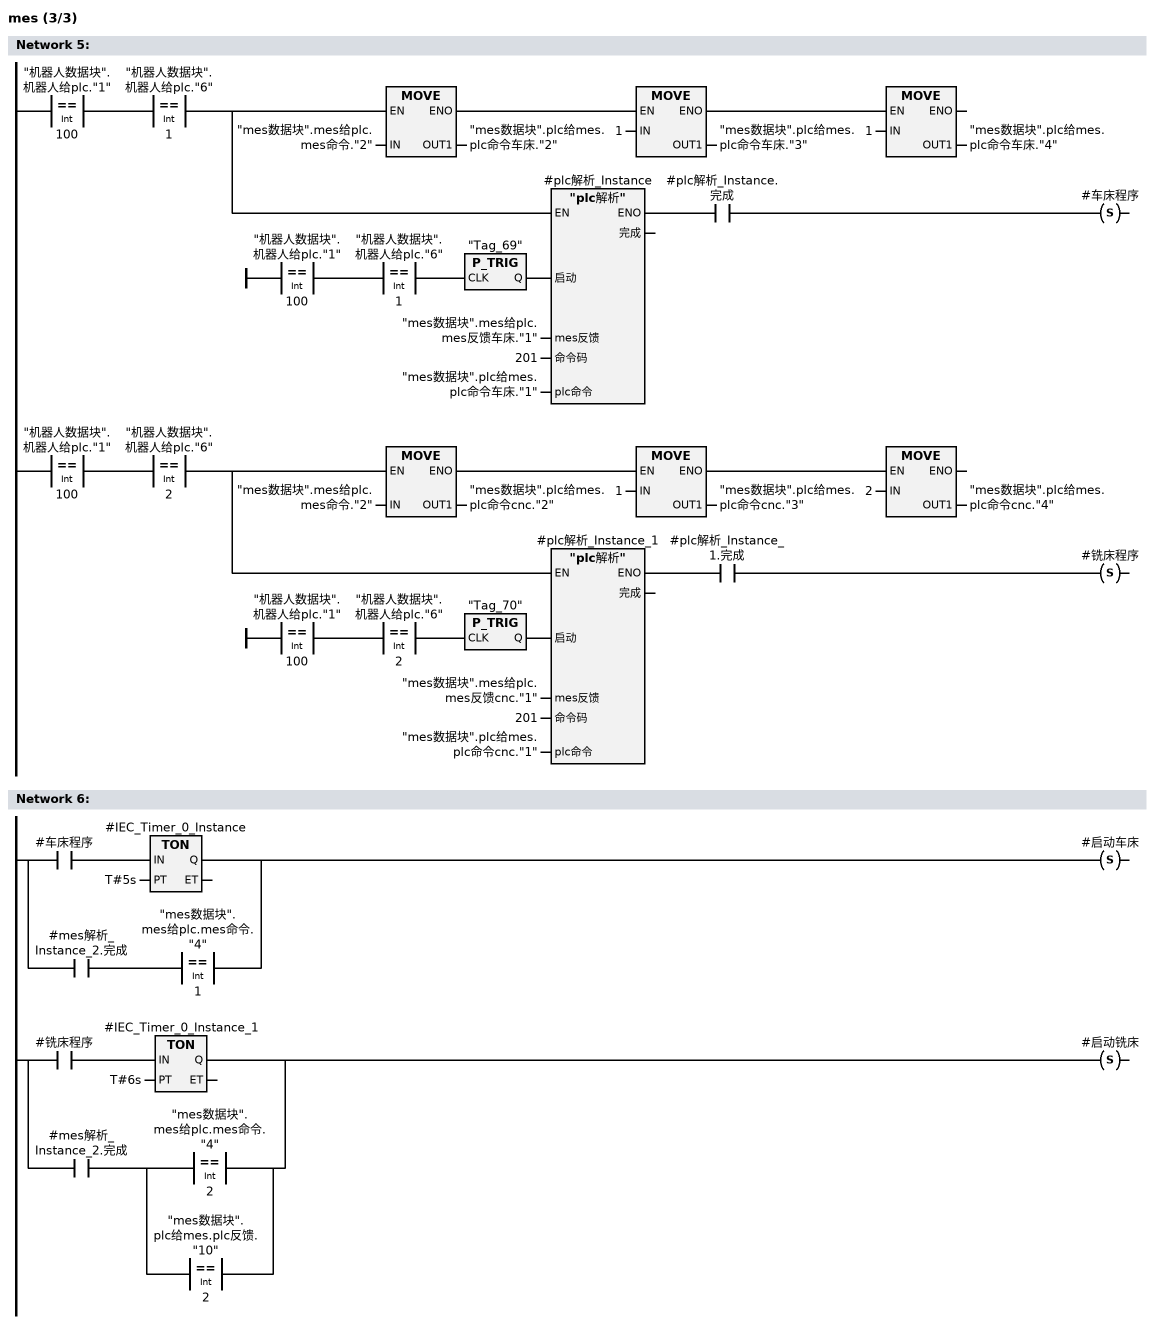
   RUNG wire#powerrail
      { S7_Templates := "SrcType := Int" } EQ_Contact(in1 := "机器人数据块".机器人给plc."1", in2 := 100)
      { S7_Templates := "SrcType := Int" } EQ_Contact(in1 := "机器人数据块".机器人给plc."6", in2 := 1)
      wire#w1
      Move(in := "mes数据块".mes给plc.mes命令."2", out1 => "mes数据块".plc给mes.plc命令车床."2")
      Move(in := 1, out1 => "mes数据块".plc给mes.plc命令车床."3")
      Move(in := 1, out1 => "mes数据块".plc给mes.plc命令车床."4")
   END_RUNG
   RUNG wire#w1
      #plc解析_Instance(启动 := wire#w2, mes反馈 := "mes数据块".mes给plc.mes反馈车床."1", 命令码 := 201, plc命令 := "mes数据块".plc给mes.plc命令车床."1", 完成 =>)
      Contact( #plc解析_Instance.完成 )
      S_Coil( #车床程序 )
   END_RUNG
   RUNG wire#powerrail
      { S7_Templates := "SrcType := Int" } EQ_Contact(in1 := "机器人数据块".机器人给plc."1", in2 := 100)
      { S7_Templates := "SrcType := Int" } EQ_Contact(in1 := "机器人数据块".机器人给plc."6", in2 := 1)
      P_Trig( "Tag_69" )
   END_RUNG wire#w2
   RUNG wire#powerrail
      { S7_Templates := "SrcType := Int" } EQ_Contact(in1 := "机器人数据块".机器人给plc."1", in2 := 100)
      { S7_Templates := "SrcType := Int" } EQ_Contact(in1 := "机器人数据块".机器人给plc."6", in2 := 2)
      wire#w3
      Move(in := "mes数据块".mes给plc.mes命令."2", out1 => "mes数据块".plc给mes.plc命令cnc."2")
      Move(in := 1, out1 => "mes数据块".plc给mes.plc命令cnc."3")
      Move(in := 2, out1 => "mes数据块".plc给mes.plc命令cnc."4")
   END_RUNG
   RUNG wire#w3
      #plc解析_Instance_1(启动 := wire#w4, mes反馈 := "mes数据块".mes给plc.mes反馈cnc."1", 命令码 := 201, plc命令 := "mes数据块".plc给mes.plc命令cnc."1", 完成 =>)
      Contact( #plc解析_Instance_1.完成 )
      S_Coil( #铣床程序 )
   END_RUNG
   RUNG wire#powerrail
      { S7_Templates := "SrcType := Int" } EQ_Contact(in1 := "机器人数据块".机器人给plc."1", in2 := 100)
      { S7_Templates := "SrcType := Int" } EQ_Contact(in1 := "机器人数据块".机器人给plc."6", in2 := 2)
      P_Trig( "Tag_70" )
   END_RUNG wire#w4
   // the same network as SCL:
   IF ("机器人数据块".机器人给plc."1" = 100) AND ("机器人数据块".机器人给plc."6" = 1) THEN
       "mes数据块".plc给mes.plc命令车床."2" := "mes数据块".mes给plc.mes命令."2";
       "mes数据块".plc给mes.plc命令车床."3" := 1;
       "mes数据块".plc给mes.plc命令车床."4" := 1;
   END_IF;
   #_w1 := ("机器人数据块".机器人给plc."1" = 100) AND ("机器人数据块".机器人给plc."6" = 1);
   #_w2 := #_w1 AND NOT "Tag_69";   // rising edge
   "Tag_69" := #_w1;
   #plc解析_Instance(EN := ("机器人数据块".机器人给plc."1" = 100) AND ("机器人数据块".机器人给plc."6" = 1),   // "plc解析"
                   启动 := #_w2,
                   mes反馈 := "mes数据块".mes给plc.mes反馈车床."1",
                   命令码 := 201,
                   plc命令 := "mes数据块".plc给mes.plc命令车床."1",
                   ENO => #_w3);
   IF #_w3 AND #plc解析_Instance.完成 THEN #车床程序 := TRUE; END_IF;
   IF ("机器人数据块".机器人给plc."1" = 100) AND ("机器人数据块".机器人给plc."6" = 2) THEN
       "mes数据块".plc给mes.plc命令cnc."2" := "mes数据块".mes给plc.mes命令."2";
       "mes数据块".plc给mes.plc命令cnc."3" := 1;
       "mes数据块".plc给mes.plc命令cnc."4" := 2;
   END_IF;
   #_w4 := ("机器人数据块".机器人给plc."1" = 100) AND ("机器人数据块".机器人给plc."6" = 2);
   #_w5 := #_w4 AND NOT "Tag_70";   // rising edge
   "Tag_70" := #_w4;
   #plc解析_Instance_1(EN := ("机器人数据块".机器人给plc."1" = 100) AND ("机器人数据块".机器人给plc."6" = 2),   // "plc解析"
                     启动 := #_w5,
                     mes反馈 := "mes数据块".mes给plc.mes反馈cnc."1",
                     命令码 := 201,
                     plc命令 := "mes数据块".plc给mes.plc命令cnc."1",
                     ENO => #_w6);
   IF #_w6 AND #plc解析_Instance_1.完成 THEN #铣床程序 := TRUE; END_IF;
END_REGION

REGION Network 6
   #IEC_Timer_0_Instance(IN := #车床程序, PT := T#5s);   // TON
   IF #IEC_Timer_0_Instance.Q OR (#mes解析_Instance_2.完成 AND ("mes数据块".mes给plc.mes命令."4" = 1)) THEN
       #启动车床 := TRUE;
   END_IF;
   #IEC_Timer_0_Instance_1(IN := #铣床程序, PT := T#6s);   // TON
   IF #IEC_Timer_0_Instance_1.Q OR (#mes解析_Instance_2.完成 AND (("mes数据块".mes给plc.mes命令."4" = 2) OR ("mes数据块".plc给mes.plc反馈."10" = 2))) THEN
       #启动铣床 := TRUE;
   END_IF;
END_REGION
END_FUNCTION_BLOCK

FUNCTION_BLOCK "机床状态"   // FB7, LAD
{ S7_Optimized_Access := 'TRUE' }
VERSION : 0.1
BEGIN

REGION Network 1
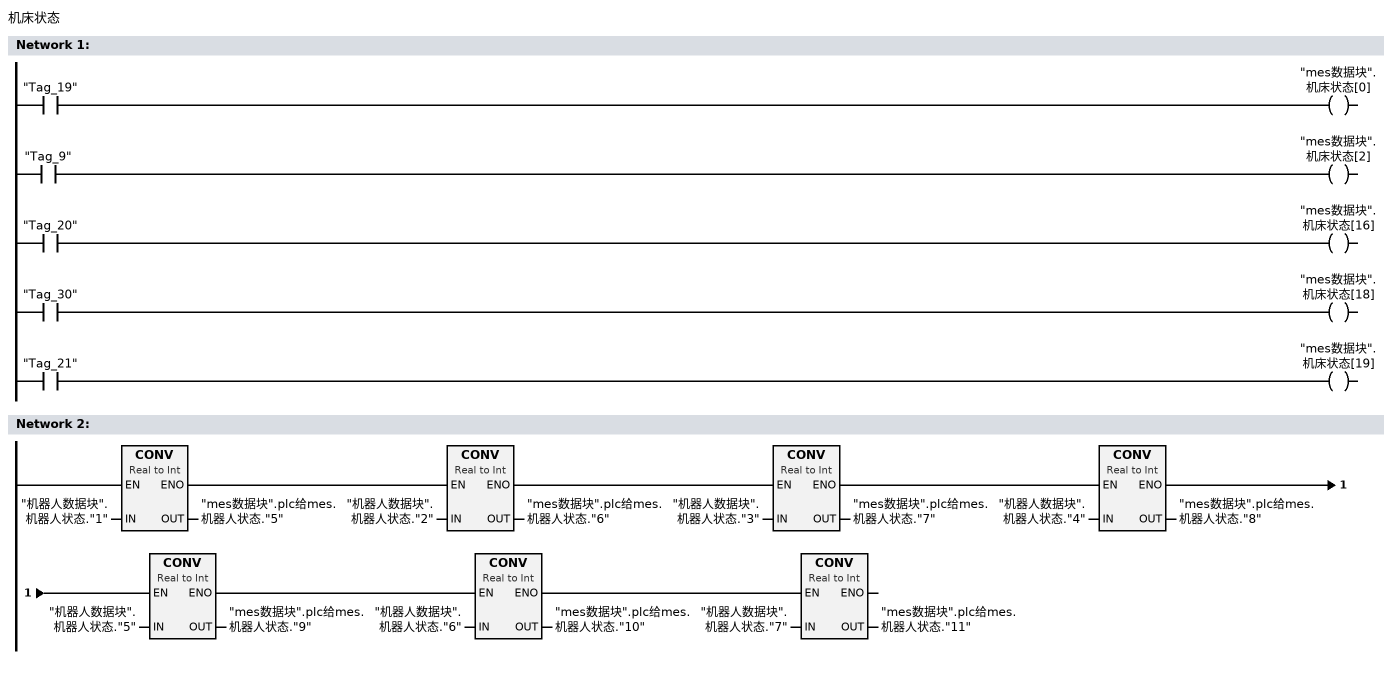
   RUNG wire#powerrail
      Contact( "Tag_19" )
      Coil( "mes数据块".机床状态[0] )
   END_RUNG
   RUNG wire#powerrail
      Contact( "Tag_9" )
      Coil( "mes数据块".机床状态[2] )
   END_RUNG
   RUNG wire#powerrail
      Contact( "Tag_20" )
      Coil( "mes数据块".机床状态[16] )
   END_RUNG
   RUNG wire#powerrail
      Contact( "Tag_30" )
      Coil( "mes数据块".机床状态[18] )
   END_RUNG
   RUNG wire#powerrail
      Contact( "Tag_21" )
      Coil( "mes数据块".机床状态[19] )
   END_RUNG
   // the same network as SCL:
   "mes数据块".机床状态[0] := "Tag_19";
   "mes数据块".机床状态[2] := "Tag_9";
   "mes数据块".机床状态[16] := "Tag_20";
   "mes数据块".机床状态[18] := "Tag_30";
   "mes数据块".机床状态[19] := "Tag_21";
END_REGION

REGION Network 2
   RUNG wire#powerrail
      { S7_Templates := "[SrcType := Real, DestType := Int]" } Convert(in := "机器人数据块".机器人状态."1", out => "mes数据块".plc给mes.机器人状态."5")
      { S7_Templates := "[SrcType := Real, DestType := Int]" } Convert(in := "机器人数据块".机器人状态."2", out => "mes数据块".plc给mes.机器人状态."6")
      { S7_Templates := "[SrcType := Real, DestType := Int]" } Convert(in := "机器人数据块".机器人状态."3", out => "mes数据块".plc给mes.机器人状态."7")
      { S7_Templates := "[SrcType := Real, DestType := Int]" } Convert(in := "机器人数据块".机器人状态."4", out => "mes数据块".plc给mes.机器人状态."8")
      { S7_Templates := "[SrcType := Real, DestType := Int]" } Convert(in := "机器人数据块".机器人状态."5", out => "mes数据块".plc给mes.机器人状态."9")
      { S7_Templates := "[SrcType := Real, DestType := Int]" } Convert(in := "机器人数据块".机器人状态."6", out => "mes数据块".plc给mes.机器人状态."10")
      { S7_Templates := "[SrcType := Real, DestType := Int]" } Convert(in := "机器人数据块".机器人状态."7", out => "mes数据块".plc给mes.机器人状态."11")
   END_RUNG
   // the same network as SCL:
   "mes数据块".plc给mes.机器人状态."5" := REAL_TO_INT("机器人数据块".机器人状态."1");
   "mes数据块".plc给mes.机器人状态."6" := REAL_TO_INT("机器人数据块".机器人状态."2");
   "mes数据块".plc给mes.机器人状态."7" := REAL_TO_INT("机器人数据块".机器人状态."3");
   "mes数据块".plc给mes.机器人状态."8" := REAL_TO_INT("机器人数据块".机器人状态."4");
   "mes数据块".plc给mes.机器人状态."9" := REAL_TO_INT("机器人数据块".机器人状态."5");
   "mes数据块".plc给mes.机器人状态."10" := REAL_TO_INT("机器人数据块".机器人状态."6");
   "mes数据块".plc给mes.机器人状态."11" := REAL_TO_INT("机器人数据块".机器人状态."7");
END_REGION
END_FUNCTION_BLOCK

FUNCTION_BLOCK "测量"   // FB8, LAD
{ S7_Optimized_Access := 'TRUE' }
VERSION : 0.1
   VAR_OUTPUT
      长度补偿 : Real;
      球半径补偿x : Real;
      球半径补偿y : Real;
      偏移补偿x : Real;
      偏移补偿y : Real;
   END_VAR
   VAR
      长度补偿整数 : Real;
      球半径补偿x_1 : Real;
      球半径补偿y_1 : Real;
      偏移补偿x_1 : Real;
      偏移补偿y_1 : Real;
      长度补偿小数 : Real;
   END_VAR
BEGIN

REGION Network 1
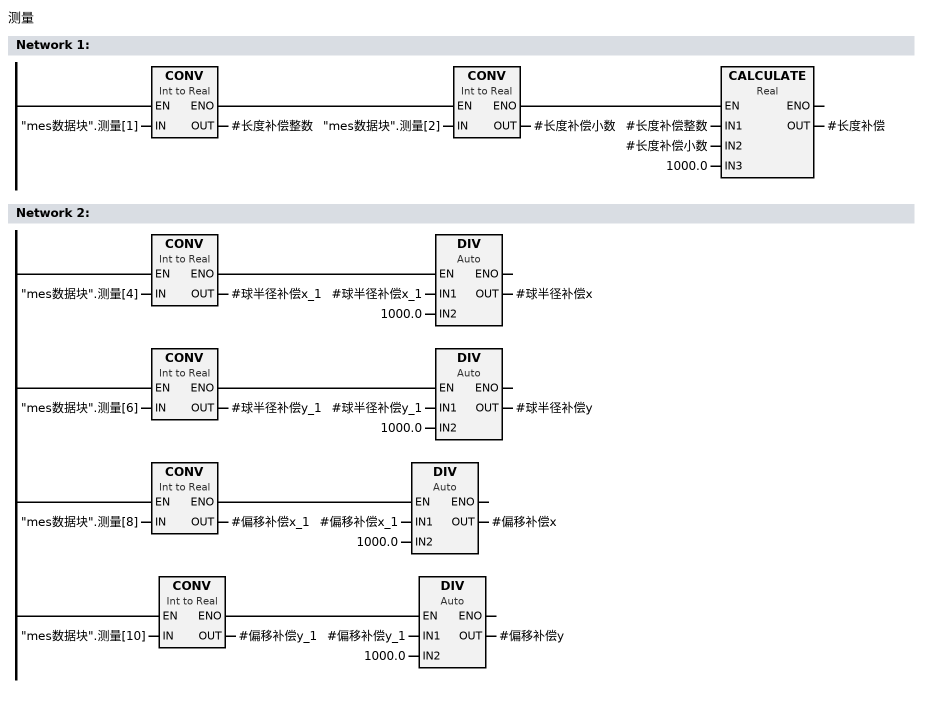
   RUNG wire#powerrail
      { S7_Templates := "[SrcType := Int, DestType := Real]" } Convert(in := "mes数据块".测量[1], out => #长度补偿整数)
      { S7_Templates := "[SrcType := Int, DestType := Real]" } Convert(in := "mes数据块".测量[2], out => #长度补偿小数)
      { S7_Templates := "SrcType := Real"; S7_Expression := "IN1+IN2/IN3" } Calculate(in1 := #长度补偿整数, in2 := #长度补偿小数, in3 := 1000.0, out => #长度补偿)
   END_RUNG
   // the same network as SCL:
   #长度补偿整数 := INT_TO_REAL("mes数据块".测量[1]);
   #长度补偿小数 := INT_TO_REAL("mes数据块".测量[2]);
   #长度补偿 := #长度补偿整数+#长度补偿小数/1000.0;
END_REGION

REGION Network 2
   RUNG wire#powerrail
      { S7_Templates := "[SrcType := Int, DestType := Real]" } Convert(in := "mes数据块".测量[4], out => #球半径补偿x_1)
      Div(in1 := #球半径补偿x_1, in2 := 1000.0, out => #球半径补偿x)
   END_RUNG
   RUNG wire#powerrail
      { S7_Templates := "[SrcType := Int, DestType := Real]" } Convert(in := "mes数据块".测量[6], out => #球半径补偿y_1)
      Div(in1 := #球半径补偿y_1, in2 := 1000.0, out => #球半径补偿y)
   END_RUNG
   RUNG wire#powerrail
      { S7_Templates := "[SrcType := Int, DestType := Real]" } Convert(in := "mes数据块".测量[8], out => #偏移补偿x_1)
      Div(in1 := #偏移补偿x_1, in2 := 1000.0, out => #偏移补偿x)
   END_RUNG
   RUNG wire#powerrail
      { S7_Templates := "[SrcType := Int, DestType := Real]" } Convert(in := "mes数据块".测量[10], out => #偏移补偿y_1)
      Div(in1 := #偏移补偿y_1, in2 := 1000.0, out => #偏移补偿y)
   END_RUNG
   // the same network as SCL:
   #球半径补偿x_1 := INT_TO_REAL("mes数据块".测量[4]);
   #球半径补偿x := #球半径补偿x_1 / 1000.0;
   #球半径补偿y_1 := INT_TO_REAL("mes数据块".测量[6]);
   #球半径补偿y := #球半径补偿y_1 / 1000.0;
   #偏移补偿x_1 := INT_TO_REAL("mes数据块".测量[8]);
   #偏移补偿x := #偏移补偿x_1 / 1000.0;
   #偏移补偿y_1 := INT_TO_REAL("mes数据块".测量[10]);
   #偏移补偿y := #偏移补偿y_1 / 1000.0;
END_REGION
END_FUNCTION_BLOCK

FUNCTION_BLOCK "有无料"   // FB10, LAD
{ S7_Optimized_Access := 'TRUE' }
VERSION : 0.1
BEGIN

REGION Network 1
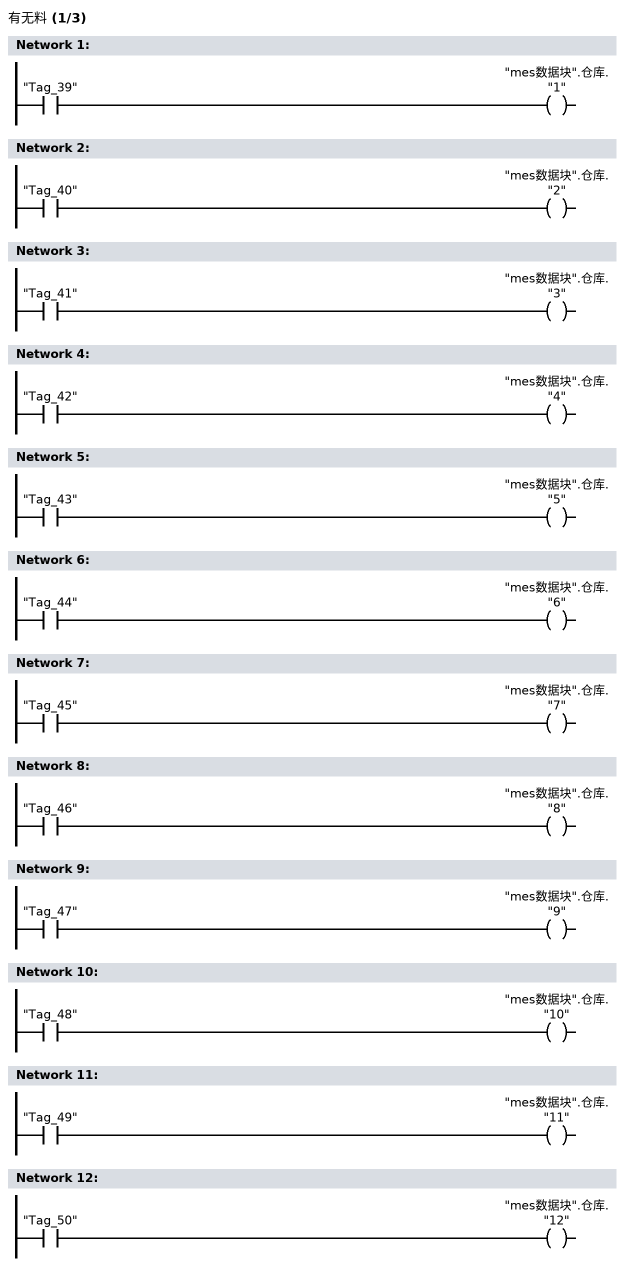
   RUNG wire#powerrail
      Contact( "Tag_39" )
      Coil( "mes数据块".仓库."1" )
   END_RUNG
   // the same network as SCL:
   "mes数据块".仓库."1" := "Tag_39";
END_REGION

REGION Network 2
   RUNG wire#powerrail
      Contact( "Tag_40" )
      Coil( "mes数据块".仓库."2" )
   END_RUNG
   // the same network as SCL:
   "mes数据块".仓库."2" := "Tag_40";
END_REGION

REGION Network 3
   RUNG wire#powerrail
      Contact( "Tag_41" )
      Coil( "mes数据块".仓库."3" )
   END_RUNG
   // the same network as SCL:
   "mes数据块".仓库."3" := "Tag_41";
END_REGION

REGION Network 4
   RUNG wire#powerrail
      Contact( "Tag_42" )
      Coil( "mes数据块".仓库."4" )
   END_RUNG
   // the same network as SCL:
   "mes数据块".仓库."4" := "Tag_42";
END_REGION

REGION Network 5
   RUNG wire#powerrail
      Contact( "Tag_43" )
      Coil( "mes数据块".仓库."5" )
   END_RUNG
   // the same network as SCL:
   "mes数据块".仓库."5" := "Tag_43";
END_REGION

REGION Network 6
   RUNG wire#powerrail
      Contact( "Tag_44" )
      Coil( "mes数据块".仓库."6" )
   END_RUNG
   // the same network as SCL:
   "mes数据块".仓库."6" := "Tag_44";
END_REGION

REGION Network 7
   RUNG wire#powerrail
      Contact( "Tag_45" )
      Coil( "mes数据块".仓库."7" )
   END_RUNG
   // the same network as SCL:
   "mes数据块".仓库."7" := "Tag_45";
END_REGION

REGION Network 8
   RUNG wire#powerrail
      Contact( "Tag_46" )
      Coil( "mes数据块".仓库."8" )
   END_RUNG
   // the same network as SCL:
   "mes数据块".仓库."8" := "Tag_46";
END_REGION

REGION Network 9
   RUNG wire#powerrail
      Contact( "Tag_47" )
      Coil( "mes数据块".仓库."9" )
   END_RUNG
   // the same network as SCL:
   "mes数据块".仓库."9" := "Tag_47";
END_REGION

REGION Network 10
   RUNG wire#powerrail
      Contact( "Tag_48" )
      Coil( "mes数据块".仓库."10" )
   END_RUNG
   // the same network as SCL:
   "mes数据块".仓库."10" := "Tag_48";
END_REGION

REGION Network 11
   RUNG wire#powerrail
      Contact( "Tag_49" )
      Coil( "mes数据块".仓库."11" )
   END_RUNG
   // the same network as SCL:
   "mes数据块".仓库."11" := "Tag_49";
END_REGION

REGION Network 12
   RUNG wire#powerrail
      Contact( "Tag_50" )
      Coil( "mes数据块".仓库."12" )
   END_RUNG
   // the same network as SCL:
   "mes数据块".仓库."12" := "Tag_50";
END_REGION

REGION Network 13
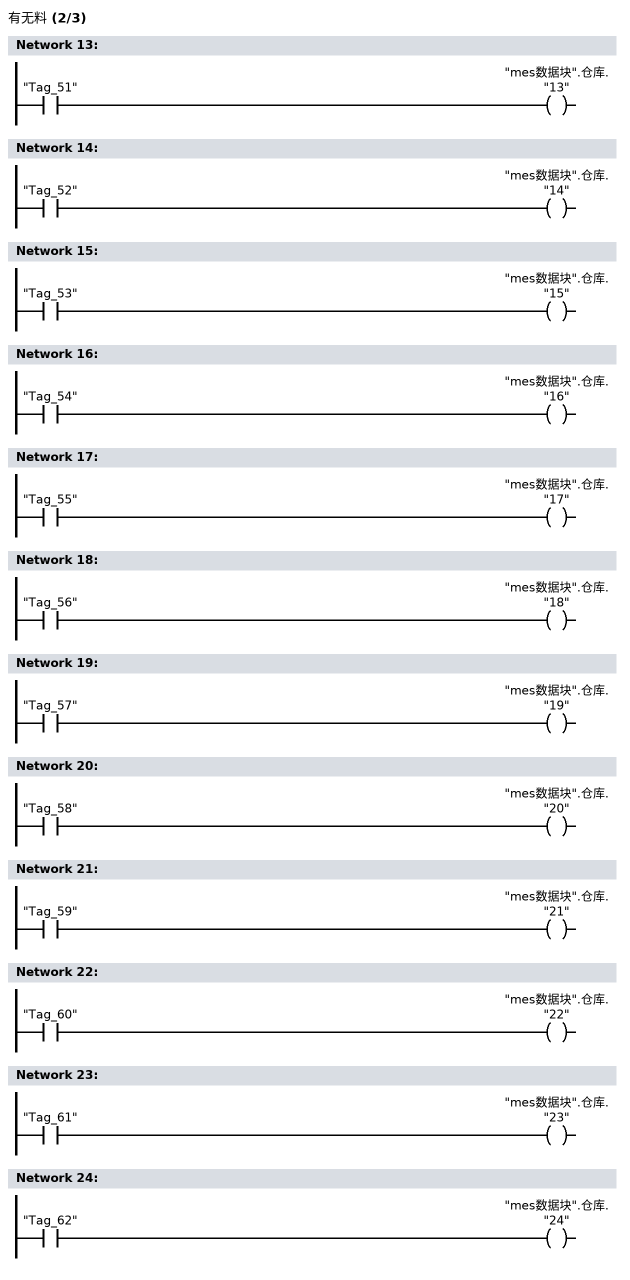
   RUNG wire#powerrail
      Contact( "Tag_51" )
      Coil( "mes数据块".仓库."13" )
   END_RUNG
   // the same network as SCL:
   "mes数据块".仓库."13" := "Tag_51";
END_REGION

REGION Network 14
   RUNG wire#powerrail
      Contact( "Tag_52" )
      Coil( "mes数据块".仓库."14" )
   END_RUNG
   // the same network as SCL:
   "mes数据块".仓库."14" := "Tag_52";
END_REGION

REGION Network 15
   RUNG wire#powerrail
      Contact( "Tag_53" )
      Coil( "mes数据块".仓库."15" )
   END_RUNG
   // the same network as SCL:
   "mes数据块".仓库."15" := "Tag_53";
END_REGION

REGION Network 16
   RUNG wire#powerrail
      Contact( "Tag_54" )
      Coil( "mes数据块".仓库."16" )
   END_RUNG
   // the same network as SCL:
   "mes数据块".仓库."16" := "Tag_54";
END_REGION

REGION Network 17
   RUNG wire#powerrail
      Contact( "Tag_55" )
      Coil( "mes数据块".仓库."17" )
   END_RUNG
   // the same network as SCL:
   "mes数据块".仓库."17" := "Tag_55";
END_REGION

REGION Network 18
   RUNG wire#powerrail
      Contact( "Tag_56" )
      Coil( "mes数据块".仓库."18" )
   END_RUNG
   // the same network as SCL:
   "mes数据块".仓库."18" := "Tag_56";
END_REGION

REGION Network 19
   RUNG wire#powerrail
      Contact( "Tag_57" )
      Coil( "mes数据块".仓库."19" )
   END_RUNG
   // the same network as SCL:
   "mes数据块".仓库."19" := "Tag_57";
END_REGION

REGION Network 20
   RUNG wire#powerrail
      Contact( "Tag_58" )
      Coil( "mes数据块".仓库."20" )
   END_RUNG
   // the same network as SCL:
   "mes数据块".仓库."20" := "Tag_58";
END_REGION

REGION Network 21
   RUNG wire#powerrail
      Contact( "Tag_59" )
      Coil( "mes数据块".仓库."21" )
   END_RUNG
   // the same network as SCL:
   "mes数据块".仓库."21" := "Tag_59";
END_REGION

REGION Network 22
   RUNG wire#powerrail
      Contact( "Tag_60" )
      Coil( "mes数据块".仓库."22" )
   END_RUNG
   // the same network as SCL:
   "mes数据块".仓库."22" := "Tag_60";
END_REGION

REGION Network 23
   RUNG wire#powerrail
      Contact( "Tag_61" )
      Coil( "mes数据块".仓库."23" )
   END_RUNG
   // the same network as SCL:
   "mes数据块".仓库."23" := "Tag_61";
END_REGION

REGION Network 24
   RUNG wire#powerrail
      Contact( "Tag_62" )
      Coil( "mes数据块".仓库."24" )
   END_RUNG
   // the same network as SCL:
   "mes数据块".仓库."24" := "Tag_62";
END_REGION

REGION Network 25
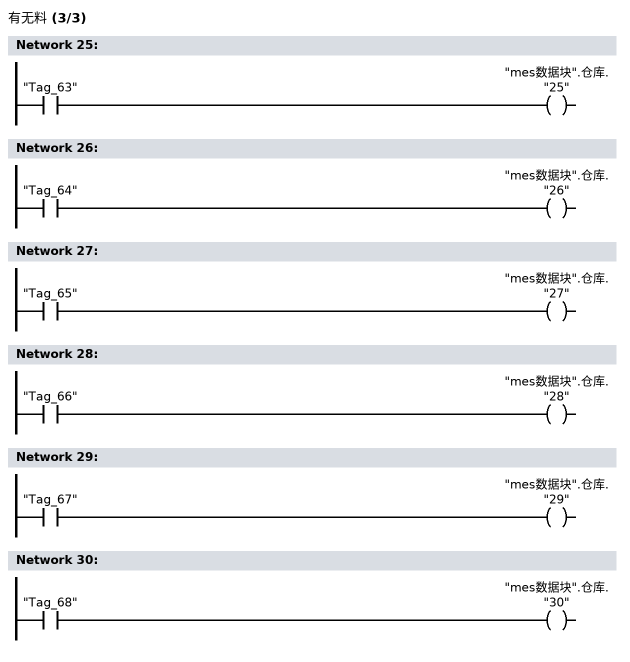
   RUNG wire#powerrail
      Contact( "Tag_63" )
      Coil( "mes数据块".仓库."25" )
   END_RUNG
   // the same network as SCL:
   "mes数据块".仓库."25" := "Tag_63";
END_REGION

REGION Network 26
   RUNG wire#powerrail
      Contact( "Tag_64" )
      Coil( "mes数据块".仓库."26" )
   END_RUNG
   // the same network as SCL:
   "mes数据块".仓库."26" := "Tag_64";
END_REGION

REGION Network 27
   RUNG wire#powerrail
      Contact( "Tag_65" )
      Coil( "mes数据块".仓库."27" )
   END_RUNG
   // the same network as SCL:
   "mes数据块".仓库."27" := "Tag_65";
END_REGION

REGION Network 28
   RUNG wire#powerrail
      Contact( "Tag_66" )
      Coil( "mes数据块".仓库."28" )
   END_RUNG
   // the same network as SCL:
   "mes数据块".仓库."28" := "Tag_66";
END_REGION

REGION Network 29
   RUNG wire#powerrail
      Contact( "Tag_67" )
      Coil( "mes数据块".仓库."29" )
   END_RUNG
   // the same network as SCL:
   "mes数据块".仓库."29" := "Tag_67";
END_REGION

REGION Network 30
   RUNG wire#powerrail
      Contact( "Tag_68" )
      Coil( "mes数据块".仓库."30" )
   END_RUNG
   // the same network as SCL:
   "mes数据块".仓库."30" := "Tag_68";
END_REGION
END_FUNCTION_BLOCK

// folder: rfid

FUNCTION_BLOCK "rfid"   // FB9, LAD
{ S7_Optimized_Access := 'TRUE' }
VERSION : 0.1
   VAR_INPUT
      仓位号 : Int;
   END_VAR
   VAR
      读 : Bool;
      写 : Bool;
      Reset_RF300_Instance : Reset_RF300;
      Read_Instance : Read;
      Write_Instance : Write;
   END_VAR
BEGIN

REGION Network 1
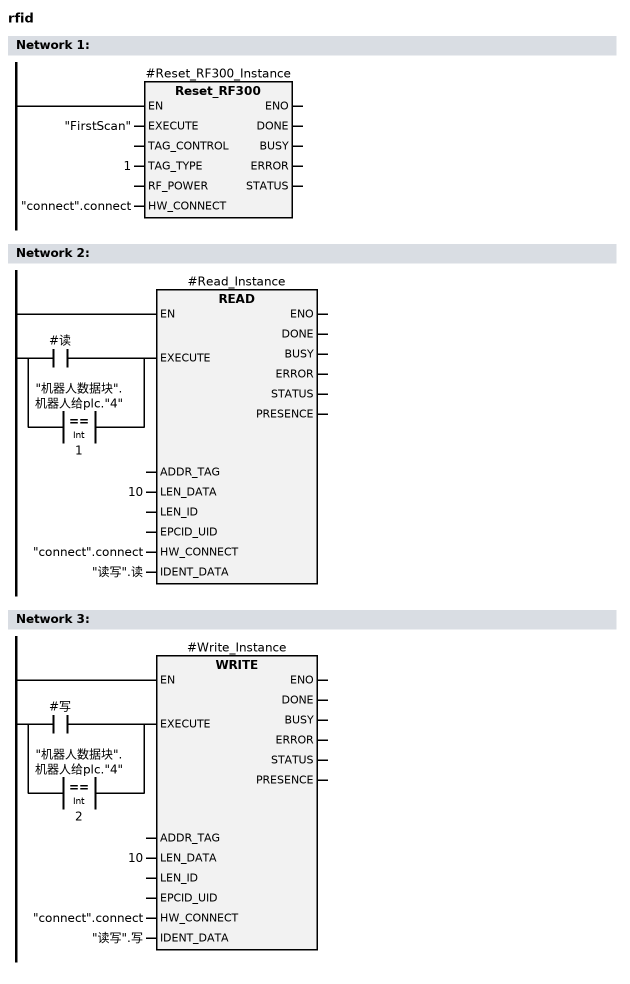
   #Reset_RF300_Instance(EXECUTE := "FirstScan", TAG_TYPE := 1, HW_CONNECT := "connect".connect);   // Reset_RF300
END_REGION

REGION Network 2
   #Read_Instance(EXECUTE := #读 OR ("机器人数据块".机器人给plc."4" = 1),   // Read
                  LEN_DATA := 10,
                  HW_CONNECT := "connect".connect,
                  IDENT_DATA := "读写".读);
END_REGION

REGION Network 3
   #Write_Instance(EXECUTE := #写 OR ("机器人数据块".机器人给plc."4" = 2),   // Write
                   LEN_DATA := 10,
                   HW_CONNECT := "connect".connect,
                   IDENT_DATA := "读写".写);
END_REGION
END_FUNCTION_BLOCK

// folder: 机床

FUNCTION_BLOCK "车床"   // FB5, LAD
{ S7_Optimized_Access := 'TRUE' }
VERSION : 0.1
   VAR_INPUT
      启动 : Bool;
   END_VAR
   VAR
      IEC_Timer_0_Instance : TON_TIME;
      IEC_Timer_0_Instance_1 : TON_TIME;
      plc解析_Instance : "plc解析";
   END_VAR
BEGIN

REGION Network 1
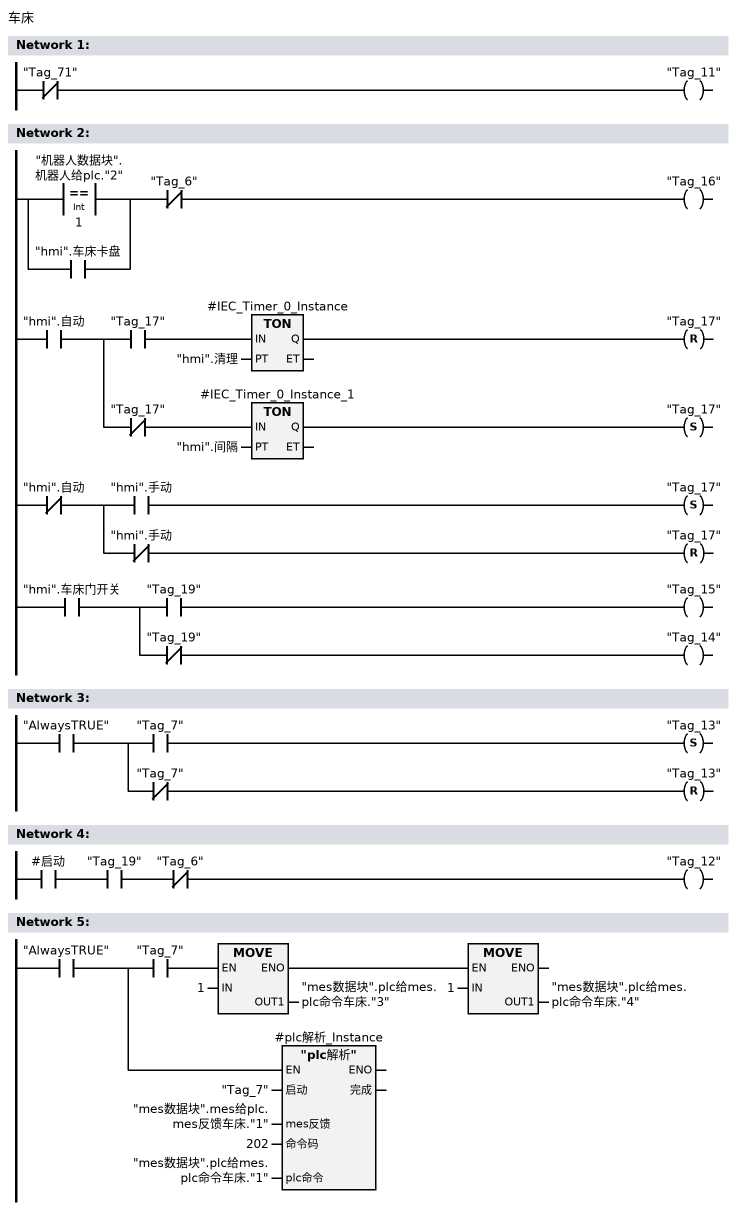
   RUNG wire#powerrail
      I_Contact( "Tag_71" )
      Coil( "Tag_11" )
   END_RUNG
   // the same network as SCL:
   "Tag_11" := NOT "Tag_71";
END_REGION

REGION Network 2
   "Tag_16" := (("机器人数据块".机器人给plc."2" = 1) OR "hmi".车床卡盘) AND NOT "Tag_6";
   #IEC_Timer_0_Instance(IN := "hmi".自动 AND "Tag_17", PT := "hmi".清理);   // TON
   IF #IEC_Timer_0_Instance.Q THEN "Tag_17" := FALSE; END_IF;
   #IEC_Timer_0_Instance_1(IN := "hmi".自动 AND NOT "Tag_17", PT := "hmi".间隔);   // TON
   IF #IEC_Timer_0_Instance_1.Q THEN "Tag_17" := TRUE; END_IF;
   IF NOT "hmi".自动 AND "hmi".手动 THEN "Tag_17" := TRUE; END_IF;
   IF NOT "hmi".自动 AND NOT "hmi".手动 THEN "Tag_17" := FALSE; END_IF;
   "Tag_15" := "hmi".车床门开关 AND "Tag_19";
   "Tag_14" := "hmi".车床门开关 AND NOT "Tag_19";
END_REGION

REGION Network 3
   RUNG wire#powerrail
      Contact( "AlwaysTRUE" )
      wire#w1
      Contact( "Tag_7" )
      S_Coil( "Tag_13" )
   END_RUNG
   RUNG wire#w1
      I_Contact( "Tag_7" )
      R_Coil( "Tag_13" )
   END_RUNG
   // the same network as SCL:
   IF "AlwaysTRUE" AND "Tag_7" THEN "Tag_13" := TRUE; END_IF;
   IF "AlwaysTRUE" AND NOT "Tag_7" THEN "Tag_13" := FALSE; END_IF;
END_REGION

REGION Network 4
   RUNG wire#powerrail
      Contact( #启动 )
      Contact( "Tag_19" )
      I_Contact( "Tag_6" )
      Coil( "Tag_12" )
   END_RUNG
   // the same network as SCL:
   "Tag_12" := #启动 AND "Tag_19" AND NOT "Tag_6";
END_REGION

REGION Network 5
   RUNG wire#powerrail
      Contact( "AlwaysTRUE" )
      wire#w1
      Contact( "Tag_7" )
      Move(in := 1, out1 => "mes数据块".plc给mes.plc命令车床."3")
      Move(in := 1, out1 => "mes数据块".plc给mes.plc命令车床."4")
   END_RUNG
   RUNG wire#w1
      #plc解析_Instance(启动 := "Tag_7", mes反馈 := "mes数据块".mes给plc.mes反馈车床."1", 命令码 := 202, plc命令 := "mes数据块".plc给mes.plc命令车床."1", 完成 =>)
   END_RUNG
   // the same network as SCL:
   IF "AlwaysTRUE" AND "Tag_7" THEN
       "mes数据块".plc给mes.plc命令车床."3" := 1;
       "mes数据块".plc给mes.plc命令车床."4" := 1;
   END_IF;
   IF "AlwaysTRUE" THEN
       #plc解析_Instance(启动 := "Tag_7",   // "plc解析"
                       mes反馈 := "mes数据块".mes给plc.mes反馈车床."1",
                       命令码 := 202,
                       plc命令 := "mes数据块".plc给mes.plc命令车床."1");
   END_IF;
END_REGION
END_FUNCTION_BLOCK

FUNCTION_BLOCK "铣床"   // FB6, LAD
{ S7_Optimized_Access := 'TRUE' }
VERSION : 0.1
   VAR_INPUT
      启动 : Bool;
   END_VAR
   VAR
      IEC_Timer_0_Instance : TON_TIME;
      IEC_Timer_0_Instance_1 : TON_TIME;
      plc解析_Instance : "plc解析";
   END_VAR
BEGIN

REGION Network 1
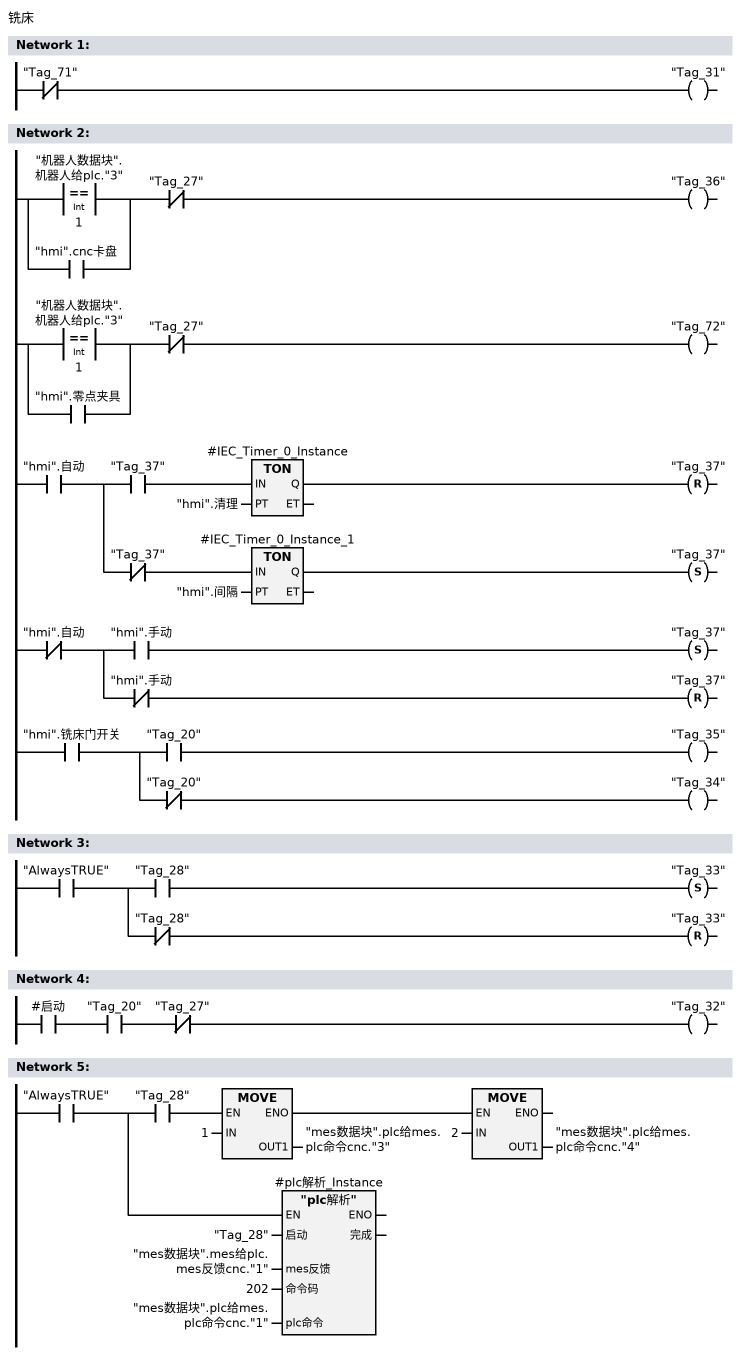
   RUNG wire#powerrail
      I_Contact( "Tag_71" )
      Coil( "Tag_31" )
   END_RUNG
   // the same network as SCL:
   "Tag_31" := NOT "Tag_71";
END_REGION

REGION Network 2
   "Tag_36" := (("机器人数据块".机器人给plc."3" = 1) OR "hmi".cnc卡盘) AND NOT "Tag_27";
   "Tag_72" := (("机器人数据块".机器人给plc."3" = 1) OR "hmi".零点夹具) AND NOT "Tag_27";
   #IEC_Timer_0_Instance(IN := "hmi".自动 AND "Tag_37", PT := "hmi".清理);   // TON
   IF #IEC_Timer_0_Instance.Q THEN "Tag_37" := FALSE; END_IF;
   #IEC_Timer_0_Instance_1(IN := "hmi".自动 AND NOT "Tag_37", PT := "hmi".间隔);   // TON
   IF #IEC_Timer_0_Instance_1.Q THEN "Tag_37" := TRUE; END_IF;
   IF NOT "hmi".自动 AND "hmi".手动 THEN "Tag_37" := TRUE; END_IF;
   IF NOT "hmi".自动 AND NOT "hmi".手动 THEN "Tag_37" := FALSE; END_IF;
   "Tag_35" := "hmi".铣床门开关 AND "Tag_20";
   "Tag_34" := "hmi".铣床门开关 AND NOT "Tag_20";
END_REGION

REGION Network 3
   RUNG wire#powerrail
      Contact( "AlwaysTRUE" )
      wire#w1
      Contact( "Tag_28" )
      S_Coil( "Tag_33" )
   END_RUNG
   RUNG wire#w1
      I_Contact( "Tag_28" )
      R_Coil( "Tag_33" )
   END_RUNG
   // the same network as SCL:
   IF "AlwaysTRUE" AND "Tag_28" THEN "Tag_33" := TRUE; END_IF;
   IF "AlwaysTRUE" AND NOT "Tag_28" THEN "Tag_33" := FALSE; END_IF;
END_REGION

REGION Network 4
   RUNG wire#powerrail
      Contact( #启动 )
      Contact( "Tag_20" )
      I_Contact( "Tag_27" )
      Coil( "Tag_32" )
   END_RUNG
   // the same network as SCL:
   "Tag_32" := #启动 AND "Tag_20" AND NOT "Tag_27";
END_REGION

REGION Network 5
   RUNG wire#powerrail
      Contact( "AlwaysTRUE" )
      wire#w1
      Contact( "Tag_28" )
      Move(in := 1, out1 => "mes数据块".plc给mes.plc命令cnc."3")
      Move(in := 2, out1 => "mes数据块".plc给mes.plc命令cnc."4")
   END_RUNG
   RUNG wire#w1
      #plc解析_Instance(启动 := "Tag_28", mes反馈 := "mes数据块".mes给plc.mes反馈cnc."1", 命令码 := 202, plc命令 := "mes数据块".plc给mes.plc命令cnc."1", 完成 =>)
   END_RUNG
   // the same network as SCL:
   IF "AlwaysTRUE" AND "Tag_28" THEN
       "mes数据块".plc给mes.plc命令cnc."3" := 1;
       "mes数据块".plc给mes.plc命令cnc."4" := 2;
   END_IF;
   IF "AlwaysTRUE" THEN
       #plc解析_Instance(启动 := "Tag_28",   // "plc解析"
                       mes反馈 := "mes数据块".mes给plc.mes反馈cnc."1",
                       命令码 := 202,
                       plc命令 := "mes数据块".plc给mes.plc命令cnc."1");
   END_IF;
END_REGION
END_FUNCTION_BLOCK

(* ===== HMI "HMI_RT_1" =====
system functions are stored by id; their names below are inferred from use
connection "HMI_连接_1": ETHERNET, S7_1200_OMS

HMI tags "默认变量表"
   "机器人数据块_机器人状态_1" : Real = PLC 机器人数据块.机器人状态.1 AT %DB2.DBD64, 1 s
   "机器人数据块_机器人状态_2" : Real = PLC 机器人数据块.机器人状态.2 AT %DB2.DBD68, 1 s
   "机器人数据块_机器人状态_3" : Real = PLC 机器人数据块.机器人状态.3 AT %DB2.DBD72, 1 s
   "机器人数据块_机器人状态_4" : Real = PLC 机器人数据块.机器人状态.4 AT %DB2.DBD76, 1 s
   "机器人数据块_机器人状态_5" : Real = PLC 机器人数据块.机器人状态.5 AT %DB2.DBD80, 1 s
   "机器人数据块_机器人状态_6" : Real = PLC 机器人数据块.机器人状态.6 AT %DB2.DBD84, 1 s
   "机器人数据块_机器人状态_7" : Real = PLC 机器人数据块.机器人状态.7 AT %DB2.DBD88, 1 s
   "hmi_机器人home位" : Bool = PLC hmi.机器人home位, 1 s
   "机器人数据块_机器人给plc_1" : Int = PLC 机器人数据块.机器人给plc.1 AT %DB2.DBW32, 1 s
   "机器人数据块_机器人状态_14" : Real = PLC 机器人数据块.机器人状态.14 AT %DB2.DBD116, 1 s
   "机器人数据块_plc给机器人_1" : Int = PLC 机器人数据块.plc给机器人.1 AT %DB2.DBW0, 1 s
   "机器人数据块_plc给机器人_2" : Int = PLC 机器人数据块.plc给机器人.2 AT %DB2.DBW2, 1 s
   "Tag_23" : Bool = PLC Tag_23 AT %Q0.5, 1 s
   "Tag_22" : Bool = PLC Tag_22 AT %Q0.4, 1 s
   "hmi_车床门开关" : Bool = PLC hmi.车床门开关, 1 s
   "hmi_车床卡盘" : Bool = PLC hmi.车床卡盘, 1 s
   "Tag_7" : Bool = PLC Tag_7 AT %I2.4, 1 s
   "Tag_3" : Bool = PLC Tag_3 AT %I2.0, 1 s
   "Tag_8" : Bool = PLC Tag_8 AT %I2.5, 1 s
   "Tag_9" : Bool = PLC Tag_9 AT %I2.6, 1 s
   "Tag_19" : Bool = PLC Tag_19 AT %I3.0, 1 s
   "Tag_28" : Bool = PLC Tag_28 AT %I4.4, 1 s
   "Tag_24" : Bool = PLC Tag_24 AT %I4.0, 1 s
   "Tag_29" : Bool = PLC Tag_29 AT %I4.5, 1 s
   "Tag_30" : Bool = PLC Tag_30 AT %I4.6, 1 s
   "Tag_21" : Bool = PLC Tag_21 AT %I5.2, 1 s
   "Tag_20" : Bool = PLC Tag_20 AT %I5.0, 1 s
   "hmi_铣床门开关" : Bool = PLC hmi.铣床门开关, 1 s
   "hmi_cnc卡盘" : Bool = PLC hmi.cnc卡盘, 1 s
   "hmi_零点夹具" : Bool = PLC hmi.零点夹具, 1 s
   "hmi_清理" : Time = PLC hmi.清理, 1 s
   "hmi_间隔" : Time = PLC hmi.间隔, 1 s
   "读写_读{4}" : Byte = PLC 读写.读[4] AT %DB6.DBB4, 1 s
   "读写_读{5}" : Byte = PLC 读写.读[5] AT %DB6.DBB5, 1 s
   "读写_读{6}" : Byte = PLC 读写.读[6] AT %DB6.DBB6, 1 s
   "读写_读{7}" : Byte = PLC 读写.读[7] AT %DB6.DBB7, 1 s
   "读写_写{4}" : Byte = PLC 读写.写[4] AT %DB6.DBB1030, 1 s
   "读写_写{5}" : Byte = PLC 读写.写[5] AT %DB6.DBB1031, 1 s
   "读写_写{6}" : Byte = PLC 读写.写[6] AT %DB6.DBB1032, 1 s
   "读写_写{7}" : Byte = PLC 读写.写[7] AT %DB6.DBB1033, 1 s
   "rfid_DB_读" : Bool = PLC rfid_DB.读, 1 s
   "rfid_DB_写" : Bool = PLC rfid_DB.写, 1 s
   "测量_DB_长度补偿" : Real = PLC 测量_DB.长度补偿, 1 s
   "测量_DB_球半径补偿x" : Real = PLC 测量_DB.球半径补偿x, 1 s
   "测量_DB_球半径补偿y" : Real = PLC 测量_DB.球半径补偿y, 1 s
   "测量_DB_偏移补偿x" : Real = PLC 测量_DB.偏移补偿x, 1 s
   "测量_DB_偏移补偿y" : Real = PLC 测量_DB.偏移补偿y, 1 s
   "mes数据块_plc给mes_plc反馈_8" : Int = PLC mes数据块.plc给mes.plc反馈.8 AT %DB1.DBW74, 1 s
   "hmi_当前仓位" : Int = PLC hmi.当前仓位, 1 s
   "hmi_种类" : Int = PLC hmi.种类, 1 s
   "机器人数据块_机器人给plc_7" : Int = PLC 机器人数据块.机器人给plc.7 AT %DB2.DBW44, 1 s
   "mes数据块_工件{1}_场次" : Int = PLC mes数据块.工件[1].场次 AT %DB1.DBW140, 1 s
   "mes数据块_工件{1}_种类" : Int = PLC mes数据块.工件[1].种类 AT %DB1.DBW142, 1 s
   "mes数据块_工件{1}_材质" : Int = PLC mes数据块.工件[1].材质 AT %DB1.DBW144, 1 s
   "mes数据块_工件{1}_状态" : Int = PLC mes数据块.工件[1].状态 AT %DB1.DBW146, 1 s
   "mes数据块_工件{2}_场次" : Int = PLC mes数据块.工件[2].场次 AT %DB1.DBW148, 1 s
   "mes数据块_工件{2}_种类" : Int = PLC mes数据块.工件[2].种类 AT %DB1.DBW150, 1 s
   "mes数据块_工件{2}_材质" : Int = PLC mes数据块.工件[2].材质 AT %DB1.DBW152, 1 s
   "mes数据块_工件{2}_状态" : Int = PLC mes数据块.工件[2].状态 AT %DB1.DBW154, 1 s
   "mes数据块_工件{3}_场次" : Int = PLC mes数据块.工件[3].场次 AT %DB1.DBW156, 1 s
   "mes数据块_工件{3}_种类" : Int = PLC mes数据块.工件[3].种类 AT %DB1.DBW158, 1 s
   "mes数据块_工件{3}_材质" : Int = PLC mes数据块.工件[3].材质 AT %DB1.DBW160, 1 s
   "mes数据块_工件{3}_状态" : Int = PLC mes数据块.工件[3].状态 AT %DB1.DBW162, 1 s
   "mes数据块_工件{4}_场次" : Int = PLC mes数据块.工件[4].场次 AT %DB1.DBW164, 1 s
   "mes数据块_工件{4}_种类" : Int = PLC mes数据块.工件[4].种类 AT %DB1.DBW166, 1 s
   "mes数据块_工件{4}_材质" : Int = PLC mes数据块.工件[4].材质 AT %DB1.DBW168, 1 s
   "mes数据块_工件{4}_状态" : Int = PLC mes数据块.工件[4].状态 AT %DB1.DBW170, 1 s
   "mes数据块_工件{5}_场次" : Int = PLC mes数据块.工件[5].场次 AT %DB1.DBW172, 1 s
   "mes数据块_工件{5}_种类" : Int = PLC mes数据块.工件[5].种类 AT %DB1.DBW174, 1 s
   "mes数据块_工件{5}_材质" : Int = PLC mes数据块.工件[5].材质 AT %DB1.DBW176, 1 s
   "mes数据块_工件{5}_状态" : Int = PLC mes数据块.工件[5].状态 AT %DB1.DBW178, 1 s
   "mes数据块_工件{6}_场次" : Int = PLC mes数据块.工件[6].场次 AT %DB1.DBW180, 1 s
   "mes数据块_工件{6}_种类" : Int = PLC mes数据块.工件[6].种类 AT %DB1.DBW182, 1 s
   "mes数据块_工件{6}_材质" : Int = PLC mes数据块.工件[6].材质 AT %DB1.DBW184, 1 s
   "mes数据块_工件{6}_状态" : Int = PLC mes数据块.工件[6].状态 AT %DB1.DBW186, 1 s
   "mes数据块_工件{7}_场次" : Int = PLC mes数据块.工件[7].场次 AT %DB1.DBW188, 1 s
   "mes数据块_工件{7}_种类" : Int = PLC mes数据块.工件[7].种类 AT %DB1.DBW190, 1 s
   "mes数据块_工件{7}_材质" : Int = PLC mes数据块.工件[7].材质 AT %DB1.DBW192, 1 s
   "mes数据块_工件{7}_状态" : Int = PLC mes数据块.工件[7].状态 AT %DB1.DBW194, 1 s
   "mes数据块_工件{8}_场次" : Int = PLC mes数据块.工件[8].场次 AT %DB1.DBW196, 1 s
   "mes数据块_工件{8}_种类" : Int = PLC mes数据块.工件[8].种类 AT %DB1.DBW198, 1 s
   "mes数据块_工件{8}_材质" : Int = PLC mes数据块.工件[8].材质 AT %DB1.DBW200, 1 s
   "mes数据块_工件{8}_状态" : Int = PLC mes数据块.工件[8].状态 AT %DB1.DBW202, 1 s
   "mes数据块_工件{9}_场次" : Int = PLC mes数据块.工件[9].场次 AT %DB1.DBW204, 1 s
   "mes数据块_工件{9}_种类" : Int = PLC mes数据块.工件[9].种类 AT %DB1.DBW206, 1 s
   "mes数据块_工件{9}_材质" : Int = PLC mes数据块.工件[9].材质 AT %DB1.DBW208, 1 s
   "mes数据块_工件{9}_状态" : Int = PLC mes数据块.工件[9].状态 AT %DB1.DBW210, 1 s
   "mes数据块_工件{10}_场次" : Int = PLC mes数据块.工件[10].场次 AT %DB1.DBW212, 1 s
   "mes数据块_工件{10}_种类" : Int = PLC mes数据块.工件[10].种类 AT %DB1.DBW214, 1 s
   "mes数据块_工件{10}_材质" : Int = PLC mes数据块.工件[10].材质 AT %DB1.DBW216, 1 s
   "mes数据块_工件{10}_状态" : Int = PLC mes数据块.工件[10].状态 AT %DB1.DBW218, 1 s
   "mes数据块_工件{11}_场次" : Int = PLC mes数据块.工件[11].场次 AT %DB1.DBW220, 1 s
   "mes数据块_工件{11}_种类" : Int = PLC mes数据块.工件[11].种类 AT %DB1.DBW222, 1 s
   "mes数据块_工件{11}_材质" : Int = PLC mes数据块.工件[11].材质 AT %DB1.DBW224, 1 s
   "mes数据块_工件{11}_状态" : Int = PLC mes数据块.工件[11].状态 AT %DB1.DBW226, 1 s
   "mes数据块_工件{12}_场次" : Int = PLC mes数据块.工件[12].场次 AT %DB1.DBW228, 1 s
   "mes数据块_工件{12}_种类" : Int = PLC mes数据块.工件[12].种类 AT %DB1.DBW230, 1 s
   "mes数据块_工件{12}_材质" : Int = PLC mes数据块.工件[12].材质 AT %DB1.DBW232, 1 s
   "mes数据块_工件{12}_状态" : Int = PLC mes数据块.工件[12].状态 AT %DB1.DBW234, 1 s
   "mes数据块_工件{13}_场次" : Int = PLC mes数据块.工件[13].场次 AT %DB1.DBW236, 1 s
   "mes数据块_工件{13}_种类" : Int = PLC mes数据块.工件[13].种类 AT %DB1.DBW238, 1 s
   "mes数据块_工件{13}_材质" : Int = PLC mes数据块.工件[13].材质 AT %DB1.DBW240, 1 s
   "mes数据块_工件{13}_状态" : Int = PLC mes数据块.工件[13].状态 AT %DB1.DBW242, 1 s
   "mes数据块_工件{14}_场次" : Int = PLC mes数据块.工件[14].场次 AT %DB1.DBW244, 1 s
   "mes数据块_工件{14}_种类" : Int = PLC mes数据块.工件[14].种类 AT %DB1.DBW246, 1 s
   "mes数据块_工件{14}_材质" : Int = PLC mes数据块.工件[14].材质 AT %DB1.DBW248, 1 s
   "mes数据块_工件{14}_状态" : Int = PLC mes数据块.工件[14].状态 AT %DB1.DBW250, 1 s
   "mes数据块_工件{15}_场次" : Int = PLC mes数据块.工件[15].场次 AT %DB1.DBW252, 1 s
   "mes数据块_工件{15}_种类" : Int = PLC mes数据块.工件[15].种类 AT %DB1.DBW254, 1 s
   "mes数据块_工件{15}_材质" : Int = PLC mes数据块.工件[15].材质 AT %DB1.DBW256, 1 s
   "mes数据块_工件{15}_状态" : Int = PLC mes数据块.工件[15].状态 AT %DB1.DBW258, 1 s
   "mes数据块_工件{16}_场次" : Int = PLC mes数据块.工件[16].场次 AT %DB1.DBW260, 1 s
   "mes数据块_工件{16}_种类" : Int = PLC mes数据块.工件[16].种类 AT %DB1.DBW262, 1 s
   "mes数据块_工件{16}_材质" : Int = PLC mes数据块.工件[16].材质 AT %DB1.DBW264, 1 s
   "mes数据块_工件{16}_状态" : Int = PLC mes数据块.工件[16].状态 AT %DB1.DBW266, 1 s
   "mes数据块_工件{17}_场次" : Int = PLC mes数据块.工件[17].场次 AT %DB1.DBW268, 1 s
   "mes数据块_工件{17}_种类" : Int = PLC mes数据块.工件[17].种类 AT %DB1.DBW270, 1 s
   "mes数据块_工件{17}_材质" : Int = PLC mes数据块.工件[17].材质 AT %DB1.DBW272, 1 s
   "mes数据块_工件{17}_状态" : Int = PLC mes数据块.工件[17].状态 AT %DB1.DBW274, 1 s
   "mes数据块_工件{18}_场次" : Int = PLC mes数据块.工件[18].场次 AT %DB1.DBW276, 1 s
   "mes数据块_工件{18}_种类" : Int = PLC mes数据块.工件[18].种类 AT %DB1.DBW278, 1 s
   "mes数据块_工件{18}_材质" : Int = PLC mes数据块.工件[18].材质 AT %DB1.DBW280, 1 s
   "mes数据块_工件{18}_状态" : Int = PLC mes数据块.工件[18].状态 AT %DB1.DBW282, 1 s
   "mes数据块_工件{19}_场次" : Int = PLC mes数据块.工件[19].场次 AT %DB1.DBW284, 1 s
   "mes数据块_工件{19}_种类" : Int = PLC mes数据块.工件[19].种类 AT %DB1.DBW286, 1 s
   "mes数据块_工件{19}_材质" : Int = PLC mes数据块.工件[19].材质 AT %DB1.DBW288, 1 s
   "mes数据块_工件{19}_状态" : Int = PLC mes数据块.工件[19].状态 AT %DB1.DBW290, 1 s
   "mes数据块_工件{20}_场次" : Int = PLC mes数据块.工件[20].场次 AT %DB1.DBW292, 1 s
   "mes数据块_工件{20}_种类" : Int = PLC mes数据块.工件[20].种类 AT %DB1.DBW294, 1 s
   "mes数据块_工件{20}_材质" : Int = PLC mes数据块.工件[20].材质 AT %DB1.DBW296, 1 s
   "mes数据块_工件{20}_状态" : Int = PLC mes数据块.工件[20].状态 AT %DB1.DBW298, 1 s
   "mes数据块_工件{21}_场次" : Int = PLC mes数据块.工件[21].场次 AT %DB1.DBW300, 1 s
   "mes数据块_工件{21}_种类" : Int = PLC mes数据块.工件[21].种类 AT %DB1.DBW302, 1 s
   "mes数据块_工件{21}_材质" : Int = PLC mes数据块.工件[21].材质 AT %DB1.DBW304, 1 s
   "mes数据块_工件{21}_状态" : Int = PLC mes数据块.工件[21].状态 AT %DB1.DBW306, 1 s
   "mes数据块_工件{22}_场次" : Int = PLC mes数据块.工件[22].场次 AT %DB1.DBW308, 1 s
   "mes数据块_工件{22}_种类" : Int = PLC mes数据块.工件[22].种类 AT %DB1.DBW310, 1 s
   "mes数据块_工件{22}_材质" : Int = PLC mes数据块.工件[22].材质 AT %DB1.DBW312, 1 s
   "mes数据块_工件{22}_状态" : Int = PLC mes数据块.工件[22].状态 AT %DB1.DBW314, 1 s
   "mes数据块_工件{23}_场次" : Int = PLC mes数据块.工件[23].场次 AT %DB1.DBW316, 1 s
   "mes数据块_工件{23}_种类" : Int = PLC mes数据块.工件[23].种类 AT %DB1.DBW318, 1 s
   "mes数据块_工件{23}_材质" : Int = PLC mes数据块.工件[23].材质 AT %DB1.DBW320, 1 s
   "mes数据块_工件{23}_状态" : Int = PLC mes数据块.工件[23].状态 AT %DB1.DBW322, 1 s
   "mes数据块_工件{24}_场次" : Int = PLC mes数据块.工件[24].场次 AT %DB1.DBW324, 1 s
   "mes数据块_工件{24}_种类" : Int = PLC mes数据块.工件[24].种类 AT %DB1.DBW326, 1 s
   "mes数据块_工件{24}_材质" : Int = PLC mes数据块.工件[24].材质 AT %DB1.DBW328, 1 s
   "mes数据块_工件{24}_状态" : Int = PLC mes数据块.工件[24].状态 AT %DB1.DBW330, 1 s
   "mes数据块_工件{25}_场次" : Int = PLC mes数据块.工件[25].场次 AT %DB1.DBW332, 1 s
   "mes数据块_工件{25}_种类" : Int = PLC mes数据块.工件[25].种类 AT %DB1.DBW334, 1 s
   "mes数据块_工件{25}_材质" : Int = PLC mes数据块.工件[25].材质 AT %DB1.DBW336, 1 s
   "mes数据块_工件{25}_状态" : Int = PLC mes数据块.工件[25].状态 AT %DB1.DBW338, 1 s
   "mes数据块_工件{26}_场次" : Int = PLC mes数据块.工件[26].场次 AT %DB1.DBW340, 1 s
   "mes数据块_工件{26}_种类" : Int = PLC mes数据块.工件[26].种类 AT %DB1.DBW342, 1 s
   "mes数据块_工件{26}_材质" : Int = PLC mes数据块.工件[26].材质 AT %DB1.DBW344, 1 s
   "mes数据块_工件{26}_状态" : Int = PLC mes数据块.工件[26].状态 AT %DB1.DBW346, 1 s
   "mes数据块_工件{27}_场次" : Int = PLC mes数据块.工件[27].场次 AT %DB1.DBW348, 1 s
   "mes数据块_工件{27}_种类" : Int = PLC mes数据块.工件[27].种类 AT %DB1.DBW350, 1 s
   "mes数据块_工件{27}_材质" : Int = PLC mes数据块.工件[27].材质 AT %DB1.DBW352, 1 s
   "mes数据块_工件{27}_状态" : Int = PLC mes数据块.工件[27].状态 AT %DB1.DBW354, 1 s
   "mes数据块_工件{28}_场次" : Int = PLC mes数据块.工件[28].场次 AT %DB1.DBW356, 1 s
   "mes数据块_工件{28}_种类" : Int = PLC mes数据块.工件[28].种类 AT %DB1.DBW358, 1 s
   "mes数据块_工件{28}_材质" : Int = PLC mes数据块.工件[28].材质 AT %DB1.DBW360, 1 s
   "mes数据块_工件{28}_状态" : Int = PLC mes数据块.工件[28].状态 AT %DB1.DBW362, 1 s
   "mes数据块_工件{29}_场次" : Int = PLC mes数据块.工件[29].场次 AT %DB1.DBW364, 1 s
   "mes数据块_工件{29}_种类" : Int = PLC mes数据块.工件[29].种类 AT %DB1.DBW366, 1 s
   "mes数据块_工件{29}_材质" : Int = PLC mes数据块.工件[29].材质 AT %DB1.DBW368, 1 s
   "mes数据块_工件{29}_状态" : Int = PLC mes数据块.工件[29].状态 AT %DB1.DBW370, 1 s
   "mes数据块_工件{30}_场次" : Int = PLC mes数据块.工件[30].场次 AT %DB1.DBW372, 1 s
   "mes数据块_工件{30}_种类" : Int = PLC mes数据块.工件[30].种类 AT %DB1.DBW374, 1 s
   "mes数据块_工件{30}_材质" : Int = PLC mes数据块.工件[30].材质 AT %DB1.DBW376, 1 s
   "mes数据块_工件{30}_状态" : Int = PLC mes数据块.工件[30].状态 AT %DB1.DBW378, 1 s
   "Tag_39" : Bool = PLC Tag_39 AT %I6.0, 1 s
   "Tag_40" : Bool = PLC Tag_40 AT %I6.1, 1 s
   "Tag_41" : Bool = PLC Tag_41 AT %I6.2, 1 s
   "Tag_42" : Bool = PLC Tag_42 AT %I6.3, 1 s
   "Tag_43" : Bool = PLC Tag_43 AT %I6.4, 1 s
   "Tag_44" : Bool = PLC Tag_44 AT %I6.5, 1 s
   "Tag_45" : Bool = PLC Tag_45 AT %I6.6, 1 s
   "Tag_46" : Bool = PLC Tag_46 AT %I6.7, 1 s
   "Tag_47" : Bool = PLC Tag_47 AT %I7.0, 1 s
   "Tag_48" : Bool = PLC Tag_48 AT %I7.1, 1 s
   "Tag_49" : Bool = PLC Tag_49 AT %I7.2, 1 s
   "Tag_50" : Bool = PLC Tag_50 AT %I7.3, 1 s
   "Tag_51" : Bool = PLC Tag_51 AT %I7.4, 1 s
   "Tag_52" : Bool = PLC Tag_52 AT %I7.5, 1 s
   "Tag_53" : Bool = PLC Tag_53 AT %I7.6, 1 s
   "Tag_54" : Bool = PLC Tag_54 AT %I8.0, 1 s
   "Tag_55" : Bool = PLC Tag_55 AT %I8.1, 1 s
   "Tag_56" : Bool = PLC Tag_56 AT %I8.2, 1 s
   "Tag_57" : Bool = PLC Tag_57 AT %I8.3, 1 s
   "Tag_58" : Bool = PLC Tag_58 AT %I8.4, 1 s
   "Tag_59" : Bool = PLC Tag_59 AT %I8.5, 1 s
   "Tag_60" : Bool = PLC Tag_60 AT %I8.6, 1 s
   "Tag_61" : Bool = PLC Tag_61 AT %I8.7, 1 s
   "Tag_62" : Bool = PLC Tag_62 AT %I9.0, 1 s
   "Tag_63" : Bool = PLC Tag_63 AT %I9.1, 1 s
   "Tag_64" : Bool = PLC Tag_64 AT %I9.2, 1 s
   "Tag_65" : Bool = PLC Tag_65 AT %I9.3, 1 s
   "Tag_66" : Bool = PLC Tag_66 AT %I9.4, 1 s
   "Tag_67" : Bool = PLC Tag_67 AT %I9.5, 1 s
   "Tag_68" : Bool = PLC Tag_68 AT %I9.6, 1 s
   "hmi_mes订单已下发" : Bool = PLC hmi.mes订单已下发, 1 s
   "机器人数据块_plc给机器人_3" : Int = PLC 机器人数据块.plc给机器人.3 AT %DB2.DBW4, 1 s
   "hmi_自动" : Bool = PLC hmi.自动, 1 s
   "hmi_手动" : Bool = PLC hmi.手动, 1 s

text list "场次": 65 'A'; 66 'B'; 67 'C'; 68 'D'; 69 'E'; 70 'A'

text list "种类": 0 '00'; 1 '01'; 2 '02'; 3 '03'; 4 '04'; 5 '05'; 6 '06'

text list "材质": 0 '铝'; 1 '钢'; 2 '0'

text list "状态": 0 '空'; 1 '毛坯'; 2 '正在加工'; 3 '合格品'; 4 '不合格品'; 5 '车床加工完成'; 6 '铣床加工完成'; 7 '00'

text list "机器人模式": 1 '手动'; 2 '自动'; 3 '外部'

text list "材质_1": 0 '铝'; 1 '钢'

text list "状态_1": 0 '空'; 1 '毛坯'; 2 '正在加工'; 3 '合格品'; 4 '不合格品'; 5 '车床加工完成'; 6 '铣床加工完成'

text list "种类_1": 3 '1'; 4 '2'; 5 '3'; 6 '4'; 7 '00'

screen "主画面" 800x480
   Button "按钮_1" at 94,29 size 230x32; TextOff 'MES与PLC交互界面'
      on Click: ActivateScreen("MES与PLC交互界面", 0)
   Button "按钮_2" at 94,84 size 230x32; TextOff 'RFID测试'
      on Click: ActivateScreen("RFID测试", 0)
   Button "按钮_3" at 94,144 size 230x32; TextOff '机床控制'
      on Click: ActivateScreen("机床控制", 0)
   Button "按钮_4" at 94,210 size 230x32; TextOff '机器人示教编程调试界面'
      on Click: ActivateScreen("机器人示教编程调试界面", 0)
   Button "按钮_5" at 94,272 size 230x32; TextOff '机器人通讯测试'
      on Click: ActivateScreen("机器人通讯测试", 0)
   Button "按钮_6" at 94,330 size 230x32; TextOff '加工中心在线测量调试界面'
      on Click: ActivateScreen("加工中心在线测量调试界面", 0)
   Button "按钮_7" at 94,384 size 230x32; TextOff '料仓信息界面'
      on Click: ActivateScreen("料仓信息界面", 0)
   Circle "圆_1" at 608,30 size 44x44
      Appearance <- "hmi_mes订单已下发"
   TextField "文本域_1" at 486,42 size 117x20; Text 'MES订单已下发'
   Button "按钮_8" at 566,116 size 96x43; TextOff '料仓盘点'
      on Release: SetTag("机器人数据块_plc给机器人_1", 0)
      on Press: SetTag("机器人数据块_plc给机器人_1", 6)

screen "机器人通讯测试" 800x480
   TextField "文本域_1" at 289,11 size 173x27; Text '机器人通讯测试'
   IOField "I/O 域_1" at 190,70 size 96x32; FormatPattern s999999999.999
      ProcessValue <- "机器人数据块_机器人状态_1"
   IOField "I/O 域_2" at 190,116 size 96x32; FormatPattern s999999999.999
      ProcessValue <- "机器人数据块_机器人状态_2"
   IOField "I/O 域_3" at 190,162 size 96x32; FormatPattern s999999999.999
      ProcessValue <- "机器人数据块_机器人状态_3"
   IOField "I/O 域_4" at 190,209 size 96x32; FormatPattern s999999999.999
      ProcessValue <- "机器人数据块_机器人状态_4"
   IOField "I/O 域_5" at 190,255 size 96x32; FormatPattern s999999999.999
      ProcessValue <- "机器人数据块_机器人状态_5"
   IOField "I/O 域_6" at 190,301 size 96x32; FormatPattern s999999999.999
      ProcessValue <- "机器人数据块_机器人状态_6"
   IOField "I/O 域_7" at 190,348 size 96x32; FormatPattern s999999999.999
      ProcessValue <- "机器人数据块_机器人状态_7"
   TextField "文本域_2" at 143,70 size 23x20; Text 'J1'
   TextField "文本域_3" at 143,116 size 23x20; Text 'J2'
   TextField "文本域_4" at 143,162 size 23x20; Text 'J3'
   TextField "文本域_5" at 143,208 size 23x20; Text 'J4'
   TextField "文本域_6" at 143,254 size 23x20; Text 'J5'
   TextField "文本域_7" at 143,300 size 23x20; Text 'J6'
   TextField "文本域_8" at 143,346 size 23x20; Text 'J7'
   TextField "文本域_9" at 311,70 size 22x20; Text '度'
   TextField "文本域_10" at 311,116 size 22x20; Text '度'
   TextField "文本域_11" at 311,162 size 22x20; Text '度'
   TextField "文本域_12" at 311,208 size 22x20; Text '度'
   TextField "文本域_13" at 311,254 size 22x20; Text '度'
   TextField "文本域_14" at 311,300 size 22x20; Text '度'
   TextField "文本域_15" at 311,346 size 39x20; Text '毫米'
   Circle "圆_1" at 613,136 size 31x31
      Appearance <- "hmi_机器人home位"
   TextField "文本域_16" at 489,141 size 109x20; Text '机器人home位'
   Circle "圆_2" at 613,194 size 31x31
      Appearance <- "机器人数据块_机器人给plc_1"
   TextField "文本域_17" at 489,199 size 99x20; Text '机器人忙/闲'
   TextField "文本域_18" at 489,254 size 90x20; Text '机器人模式'
   SymbolicIOField "符号 I/O 域_1" at 598,252 size 93x32; TextOff '0'; TextOn '1'; TextList "机器人模式"
      ProcessValue <- "机器人数据块_机器人状态_14"
   Button "按钮_1" at 14,437 size 104x32; TextOff '主画面'
      on Click: ActivateScreen("主画面", 0)

screen "机器人示教编程调试界面" 800x480
   TextField "文本域_1" at 272,15 size 269x27; Text '机器人示教编程调试界面'
   Button "按钮_1" at 53,66 size 96x43; TextOff '料仓取料'
      on Press: SetTag("机器人数据块_plc给机器人_1", 1)
      on Release: SetTag("机器人数据块_plc给机器人_1", 0)
   Button "按钮_2" at 53,138 size 96x43; TextOff '车床放料'
      on Release: SetTag("机器人数据块_plc给机器人_1", 0)
      on Press: SetTag("机器人数据块_plc给机器人_1", 11)
   Button "按钮_3" at 53,210 size 96x43; TextOff '车床取料'
      on Release: SetTag("机器人数据块_plc给机器人_1", 0)
      on Press: SetTag("机器人数据块_plc给机器人_1", 12)
   Button "按钮_4" at 589,66 size 124x43; TextOff '料仓放料'
      on Release: SetTag("机器人数据块_plc给机器人_1", 0)
      on Press: SetTag("机器人数据块_plc给机器人_1", 2)
   Button "按钮_5" at 589,138 size 124x43; TextOff '加工中心放料'
      on Release: SetTag("机器人数据块_plc给机器人_1", 0)
      on Press: SetTag("机器人数据块_plc给机器人_1", 31)
   Button "按钮_6" at 589,210 size 124x43; TextOff '加工中心取料'
      on Release: SetTag("机器人数据块_plc给机器人_1", 0)
      on Press: SetTag("机器人数据块_plc给机器人_1", 32)
   Button "按钮_7" at 309,210 size 155x43; TextOff '车床到加工中心'
      on Release: SetTag("机器人数据块_plc给机器人_1", 0)
      on Press: SetTag("机器人数据块_plc给机器人_1", 21)
   TextField "文本域_2" at 340,67 size 90x20; Text '指定仓位号'
   TextField "文本域_3" at 198,116 size 73x20; Text '料仓行号'
   IOField "I/O 域_1" at 272,113 size 48x32; FormatPattern 99
      ProcessValue <- "机器人数据块_plc给机器人_2"
   TextField "文本域_4" at 405,119 size 73x20; Text '料仓列号'
   IOField "I/O 域_2" at 482,114 size 48x32; FormatPattern 99
      ProcessValue <- "机器人数据块_plc给机器人_3"
   Button "按钮_8" at 239,291 size 117x41; TextOff '机器人暂停'
      on Press: SetBit("Tag_23")
      on Release: ResetBit("Tag_23")
   Button "按钮_9" at 413,291 size 117x41; TextOff '机器人继续'
      on Release: ResetBit("Tag_22")
      on Press: SetBit("Tag_22")
   Button "按钮_10" at 12,444 size 120x32; TextOff '主画面'
      on Click: ActivateScreen("主画面", 0)

screen "机床控制" 800x480
   TextField "文本域_1" at 101,15 size 93x25; Text '车床控制'
   Button "按钮_1" at 26,95 size 119x38; TextOff '车床门开关'
      on Press: SetBit("hmi_车床门开关")
      on Release: ResetBit("hmi_车床门开关")
   Button "按钮_2" at 26,168 size 119x35; TextOff '车床卡盘松紧'
      on Press: InvertBit("hmi_车床卡盘")
   Circle "圆_1" at 295,56 size 31x31
      Appearance <- "Tag_7"
   TextField "文本域_2" at 169,60 size 107x20; Text '车床加工完成'
   Circle "圆_2" at 295,102 size 31x31
      Appearance <- "Tag_3"
   TextField "文本域_3" at 169,106 size 73x20; Text '车床联机'
   Circle "圆_3" at 295,148 size 31x31
      Appearance <- "Tag_8"
   TextField "文本域_4" at 169,152 size 73x20; Text '车床报警'
   Circle "圆_4" at 295,194 size 31x31
      Appearance <- "Tag_9"
   TextField "文本域_5" at 169,198 size 107x20; Text '车床卡盘松紧'
   Circle "圆_5" at 295,240 size 31x31
      Appearance <- "Tag_19"
   TextField "文本域_6" at 169,244 size 90x20; Text '车床门状态'
   Circle "圆_6" at 739,60 size 31x31
      Appearance <- "Tag_28"
   TextField "文本域_7" at 585,65 size 141x20; Text '加工中心加工完成'
   Circle "圆_7" at 739,101 size 31x31
      Appearance <- "Tag_24"
   TextField "文本域_8" at 585,106 size 107x20; Text '加工中心联机'
   Circle "圆_8" at 739,142 size 31x31
      Appearance <- "Tag_29"
   TextField "文本域_9" at 585,147 size 107x20; Text '加工中心报警'
   Circle "圆_9" at 739,183 size 31x31
      Appearance <- "Tag_30"
   TextField "文本域_10" at 585,188 size 73x20; Text '虎钳松紧'
   Circle "圆_10" at 739,224 size 31x31
      Appearance <- "Tag_21"
   TextField "文本域_11" at 585,229 size 141x20; Text '零点定位夹具松紧'
   Circle "圆_11" at 739,265 size 31x31
      Appearance <- "Tag_20"
   TextField "文本域_12" at 585,270 size 124x20; Text '加工中心门状态'
   Button "按钮_3" at 379,102 size 146x38; TextOff '加工中心门开关'
      on Release: ResetBit("hmi_铣床门开关")
      on Press: SetBit("hmi_铣床门开关")
   Button "按钮_4" at 379,154 size 146x32; TextOff '虎钳松紧'
      on Press: InvertBit("hmi_cnc卡盘")
   Button "按钮_5" at 376,200 size 146x32; TextOff '零点定位夹具松'
      on Press: InvertBit("hmi_零点夹具")
   Button "按钮_6" at 379,245 size 146x32; TextOff '零点定位夹具紧'
      on Press: InvertBit("hmi_零点夹具")
   Button "按钮_7" at 39,295 size 146x38; TextOff '相机自动清理'
      on Press: InvertBit("hmi_自动")
   Button "按钮_8" at 241,296 size 146x38; TextOff '相机手动清理'
      on Release: ResetBit("hmi_手动")
      on Press: SetBit("hmi_手动")
   IOField "I/O 域_1" at 81,352 size 96x32; FormatPattern 9999
      ProcessValue <- "hmi_清理"
   IOField "I/O 域_2" at 291,352 size 96x32; FormatPattern 9999
      ProcessValue <- "hmi_间隔"
   TextField "文本域_13" at 394,357 size 14x20; Text 'S'
   TextField "文本域_14" at 184,359 size 14x20; Text 'S'
   TextField "文本域_15" at 1,357 size 90x20; Text '吹气时间：'
   TextField "文本域_16" at 209,357 size 90x20; Text '间歇时间：'
   Button "按钮_9" at 6,441 size 88x32; TextOff '主画面'
      on Click: ActivateScreen("主画面", 0)
   Button "按钮_10" at 104,441 size 99x32; TextOff 'RFID测试'
      on Click: ActivateScreen("RFID测试", 0)
   Button "按钮_11" at 212,441 size 106x32; TextOff '机器人示教'; TextOn '机器人示教编程调试界面'
      on Click: ActivateScreen("机器人示教编程调试界面", 0)
   Button "按钮_12" at 330,441 size 102x32; TextOff '机器人通讯'; TextOn '机器人通讯测试'
      on Click: ActivateScreen("机器人通讯测试", 0)
   Button "按钮_13" at 442,441 size 96x32; TextOff '测头标定'; TextOn '加工中心在线测量调试界面'
      on Click: ActivateScreen("加工中心在线测量调试界面", 0)
   Button "按钮_14" at 547,441 size 105x32; TextOff '料仓监测'; TextOn '料仓信息界面'
      on Click: ActivateScreen("料仓信息界面", 0)
   Button "按钮_15" at 665,441 size 94x32; TextOff 'MES交互'; TextOn 'MES与PLC交互界面'
      on Click: ActivateScreen("MES与PLC交互界面", 0)

screen "RFID测试" 800x480
   TextField "文本域_1" at 324,11 size 153x27; Text 'RFID读写控制'
   TextField "文本域_2" at 94,52 size 71x25; Text '读数据'
   TextField "文本域_3" at 54,90 size 14x20; Text '1'
   TextField "文本域_4" at 54,194 size 14x20; Text '2'
   TextField "文本域_5" at 54,299 size 14x20; Text '3'
   TextField "文本域_6" at 54,404 size 14x20; Text '4'
   SymbolicIOField "符号 I/O 域_1" at 75,90 size 130x37; TextOff '0'; TextOn '1'; TextList "场次"
      ProcessValue <- "读写_读{4}"
   SymbolicIOField "符号 I/O 域_2" at 75,194 size 130x37; TextOn '1'; TextOff '0'; TextList "种类"
      ProcessValue <- "读写_读{5}"
   SymbolicIOField "符号 I/O 域_3" at 75,298 size 130x37; TextOn '1'; TextOff '0'; TextList "材质"
      ProcessValue <- "读写_读{6}"
   SymbolicIOField "符号 I/O 域_4" at 75,397 size 130x37; TextOn '1'; TextOff '0'; TextList "状态"
      ProcessValue <- "读写_读{7}"
   TextField "文本域_7" at 353,52 size 71x25; Text '写数据'
   TextField "文本域_8" at 313,90 size 14x20; Text '1'
   TextField "文本域_9" at 313,194 size 14x20; Text '2'
   TextField "文本域_10" at 313,299 size 14x20; Text '3'
   TextField "文本域_11" at 313,404 size 14x20; Text '4'
   SymbolicIOField "符号 I/O 域_5" at 337,90 size 130x37; TextOn '1'; TextOff '0'; TextList "场次"
      ProcessValue <- "读写_写{4}"
   SymbolicIOField "符号 I/O 域_6" at 337,194 size 130x37; TextOn '1'; TextOff '0'; TextList "种类"
      ProcessValue <- "读写_写{5}"
   SymbolicIOField "符号 I/O 域_7" at 337,298 size 130x37; TextOn '1'; TextOff '0'; TextList "材质"
      ProcessValue <- "读写_写{6}"
   SymbolicIOField "符号 I/O 域_8" at 337,402 size 130x37; TextOn '1'; TextOff '0'; TextList "状态"
      ProcessValue <- "读写_写{7}"
   TextField "文本域_12" at 622,52 size 49x25; Text '操作'
   Button "按钮_1" at 584,117 size 110x39; TextOff '初始化'
      on Press: SetTag("读写_读{4}", 0); SetTag("读写_读{5}", 0); SetTag("读写_读{6}", 0); SetTag("读写_读{7}", 0); SetTag("读写_写{4}", 0); SetTag("读写_写{5}", 0); SetTag("读写_写{6}", 0); SetTag("读写_写{7}", 0)
   Button "按钮_3" at 584,214 size 110x39; TextOff '读卡'
      on Press: SetTag("机器人数据块_plc给机器人_1", 3)
      on Release: SetTag("机器人数据块_plc给机器人_1", 0)
   Button "按钮_2" at 584,323 size 110x39; TextOff '写卡'
      on Press: SetTag("机器人数据块_plc给机器人_1", 4)
      on Release: SetTag("机器人数据块_plc给机器人_1", 0)
   Button "按钮_4" at 596,6 size 192x32; TextOff 'Text'; TextOn '主画面'
      on Click: ActivateScreen("主画面", 0)

screen "加工中心在线测量调试界面" 800x480
   TextField "文本域_1" at 249,7 size 293x27; Text '加工中心在线测量调试界面'
   TextField "文本域_2" at 159,66 size 137x25; Text '测头长度补偿'
   TextField "文本域_3" at 147,129 size 149x25; Text '测头偏移补偿X'
   TextField "文本域_4" at 147,193 size 149x25; Text '测头偏移补偿Y'
   TextField "文本域_5" at 125,257 size 171x25; Text '测头球半径补偿X'
   TextField "文本域_6" at 125,321 size 171x25; Text '测头球半径补偿Y'
   IOField "I/O 域_1" at 323,66 size 149x32; FormatPattern 99.999
      ProcessValue <- "测量_DB_长度补偿"
   IOField "I/O 域_2" at 323,257 size 149x32; FormatPattern 99.999
      ProcessValue <- "测量_DB_球半径补偿x"
   IOField "I/O 域_3" at 323,321 size 149x32; FormatPattern 99.999
      ProcessValue <- "测量_DB_球半径补偿y"
   IOField "I/O 域_4" at 323,129 size 149x32; FormatPattern 99.999
      ProcessValue <- "测量_DB_偏移补偿x"
   IOField "I/O 域_5" at 323,193 size 149x32; FormatPattern 99.999
      ProcessValue <- "测量_DB_偏移补偿y"
   TextField "文本域_7" at 512,66 size 29x25; Text 'mm'
   TextField "文本域_8" at 512,129 size 29x25; Text 'mm'
   TextField "文本域_9" at 512,192 size 29x25; Text 'mm'
   TextField "文本域_10" at 512,255 size 29x25; Text 'mm'
   TextField "文本域_11" at 512,318 size 29x25; Text 'mm'
   Button "按钮_1" at 599,66 size 179x37; TextOff '测量数据采集'
      on Press: SetTag("mes数据块_plc给mes_plc反馈_8", 106)
      on Release: SetTag("mes数据块_plc给mes_plc反馈_8", 0)
   Button "按钮_2" at 5,444 size 98x32; TextOff '主画面'
      on Click: ActivateScreen("主画面", 0)

screen "MES与PLC交互界面" 800x480
   TextField "文本域_1" at 295,15 size 187x25; Text 'MES与PLC交互界面'
   TextField "文本域_2" at 104,65 size 225x25; Text '当前执行中的工单状态'
   IOField "I/O 域_1" at 114,151 size 96x32; FormatPattern 99
      ProcessValue <- "hmi_当前仓位"
   TextField "文本域_3" at 109,122 size 117x19; Text '工件所在库位号'
   TextField "文本域_4" at 293,122 size 69x19; Text '工件种类'
   TextField "文本域_5" at 477,122 size 101x19; Text '工件加工状态'
   SymbolicIOField "符号 I/O 域_6" at 291,151 size 101x32; TextOn '1'; TextOff '0'; TextList "种类_1"
      ProcessValue <- "hmi_种类"
   SymbolicIOField "符号 I/O 域_8" at 482,151 size 145x32; TextOn '1'; TextOff '0'; TextList "状态_1"
      ProcessValue <- "机器人数据块_机器人给plc_7"
   Button "按钮_1" at 10,445 size 100x32; TextOff '主画面'
      on Click: ActivateScreen("主画面", 0)

screen "料仓信息界面" 800x480
   TextField "文本域_1" at 292,447 size 149x27; Text '料仓信息界面'
   TextField "文本域_2" at 10,8 size 44x16; Text '仓位号'
   TextField "文本域_3" at 17,36 size 31x16; Text '场次'
   TextField "文本域_4" at 16,69 size 31x16; Text '种类'
   TextField "文本域_5" at 16,107 size 31x16; Text '材质'
   TextField "文本域_6" at 16,142 size 31x16; Text '状态'
   SymbolicIOField "符号 I/O 域_1" at 57,32 size 40x27; TextOff '0'; TextOn '1'; TextList "场次"
      ProcessValue <- "mes数据块_工件{1}_场次"
   SymbolicIOField "符号 I/O 域_2" at 57,65 size 40x27; TextOn '1'; TextOff '0'; TextList "种类"
      ProcessValue <- "mes数据块_工件{1}_种类"
   SymbolicIOField "符号 I/O 域_3" at 57,103 size 40x27; TextOn '1'; TextOff '0'; TextList "材质_1"
      ProcessValue <- "mes数据块_工件{1}_材质"
   SymbolicIOField "符号 I/O 域_4" at 57,138 size 40x27; TextOn '1'; TextOff '0'; TextList "状态_1"
      ProcessValue <- "mes数据块_工件{1}_状态"
   SymbolicIOField "符号 I/O 域_5" at 103,32 size 40x27; TextOn '1'; TextOff '0'; TextList "场次"
      ProcessValue <- "mes数据块_工件{2}_场次"
   SymbolicIOField "符号 I/O 域_6" at 103,65 size 40x27; TextOn '1'; TextOff '0'; TextList "种类"
      ProcessValue <- "mes数据块_工件{2}_种类"
   SymbolicIOField "符号 I/O 域_7" at 103,103 size 40x27; TextOn '1'; TextOff '0'; TextList "材质_1"
      ProcessValue <- "mes数据块_工件{2}_材质"
   SymbolicIOField "符号 I/O 域_8" at 103,138 size 40x27; TextOn '1'; TextOff '0'; TextList "状态_1"
      ProcessValue <- "mes数据块_工件{2}_状态"
   SymbolicIOField "符号 I/O 域_9" at 149,32 size 40x27; TextOn '1'; TextOff '0'; TextList "场次"
      ProcessValue <- "mes数据块_工件{3}_场次"
   SymbolicIOField "符号 I/O 域_10" at 149,65 size 40x27; TextOn '1'; TextOff '0'; TextList "种类"
      ProcessValue <- "mes数据块_工件{3}_种类"
   SymbolicIOField "符号 I/O 域_11" at 149,103 size 40x27; TextOn '1'; TextOff '0'; TextList "材质_1"
      ProcessValue <- "mes数据块_工件{3}_材质"
   SymbolicIOField "符号 I/O 域_12" at 149,138 size 40x27; TextOn '1'; TextOff '0'; TextList "状态_1"
      ProcessValue <- "mes数据块_工件{3}_状态"
   SymbolicIOField "符号 I/O 域_13" at 195,32 size 40x27; TextOn '1'; TextOff '0'; TextList "场次"
      ProcessValue <- "mes数据块_工件{4}_场次"
   SymbolicIOField "符号 I/O 域_14" at 195,65 size 40x27; TextOn '1'; TextOff '0'; TextList "种类"
      ProcessValue <- "mes数据块_工件{4}_种类"
   SymbolicIOField "符号 I/O 域_15" at 195,103 size 40x27; TextOn '1'; TextOff '0'; TextList "材质_1"
      ProcessValue <- "mes数据块_工件{4}_材质"
   SymbolicIOField "符号 I/O 域_16" at 195,138 size 40x27; TextOn '1'; TextOff '0'; TextList "状态_1"
      ProcessValue <- "mes数据块_工件{4}_状态"
   SymbolicIOField "符号 I/O 域_17" at 241,32 size 40x27; TextOn '1'; TextOff '0'; TextList "场次"
      ProcessValue <- "mes数据块_工件{5}_场次"
   SymbolicIOField "符号 I/O 域_18" at 241,65 size 40x27; TextOn '1'; TextOff '0'; TextList "种类"
      ProcessValue <- "mes数据块_工件{5}_种类"
   SymbolicIOField "符号 I/O 域_19" at 241,103 size 40x27; TextOn '1'; TextOff '0'; TextList "材质_1"
      ProcessValue <- "mes数据块_工件{5}_材质"
   SymbolicIOField "符号 I/O 域_20" at 241,138 size 40x27; TextOn '1'; TextOff '0'; TextList "状态_1"
      ProcessValue <- "mes数据块_工件{5}_状态"
   SymbolicIOField "符号 I/O 域_21" at 287,32 size 40x27; TextOn '1'; TextOff '0'; TextList "场次"
      ProcessValue <- "mes数据块_工件{6}_场次"
   SymbolicIOField "符号 I/O 域_22" at 287,65 size 40x27; TextOn '1'; TextOff '0'; TextList "种类"
      ProcessValue <- "mes数据块_工件{6}_种类"
   SymbolicIOField "符号 I/O 域_23" at 287,103 size 40x27; TextOn '1'; TextOff '0'; TextList "材质_1"
      ProcessValue <- "mes数据块_工件{6}_材质"
   SymbolicIOField "符号 I/O 域_24" at 287,138 size 40x27; TextOn '1'; TextOff '0'; TextList "状态_1"
      ProcessValue <- "mes数据块_工件{6}_状态"
   SymbolicIOField "符号 I/O 域_25" at 333,32 size 40x27; TextOn '1'; TextOff '0'; TextList "场次"
      ProcessValue <- "mes数据块_工件{7}_场次"
   SymbolicIOField "符号 I/O 域_26" at 333,65 size 40x27; TextOn '1'; TextOff '0'; TextList "种类"
      ProcessValue <- "mes数据块_工件{7}_种类"
   SymbolicIOField "符号 I/O 域_27" at 333,103 size 40x27; TextOn '1'; TextOff '0'; TextList "材质_1"
      ProcessValue <- "mes数据块_工件{7}_材质"
   SymbolicIOField "符号 I/O 域_28" at 333,138 size 40x27; TextOn '1'; TextOff '0'; TextList "状态_1"
      ProcessValue <- "mes数据块_工件{7}_状态"
   SymbolicIOField "符号 I/O 域_29" at 379,32 size 40x27; TextOn '1'; TextOff '0'; TextList "场次"
      ProcessValue <- "mes数据块_工件{8}_场次"
   SymbolicIOField "符号 I/O 域_30" at 379,65 size 40x27; TextOn '1'; TextOff '0'; TextList "种类"
      ProcessValue <- "mes数据块_工件{8}_种类"
   SymbolicIOField "符号 I/O 域_31" at 379,103 size 40x27; TextOn '1'; TextOff '0'; TextList "材质_1"
      ProcessValue <- "mes数据块_工件{8}_材质"
   SymbolicIOField "符号 I/O 域_32" at 379,138 size 40x27; TextOn '1'; TextOff '0'; TextList "状态_1"
      ProcessValue <- "mes数据块_工件{8}_状态"
   SymbolicIOField "符号 I/O 域_33" at 425,32 size 40x27; TextOn '1'; TextOff '0'; TextList "场次"
      ProcessValue <- "mes数据块_工件{9}_场次"
   SymbolicIOField "符号 I/O 域_34" at 425,65 size 40x27; TextOn '1'; TextOff '0'; TextList "种类"
      ProcessValue <- "mes数据块_工件{9}_种类"
   SymbolicIOField "符号 I/O 域_35" at 425,103 size 40x27; TextOn '1'; TextOff '0'; TextList "材质_1"
      ProcessValue <- "mes数据块_工件{9}_材质"
   SymbolicIOField "符号 I/O 域_36" at 425,138 size 40x27; TextOn '1'; TextOff '0'; TextList "状态_1"
      ProcessValue <- "mes数据块_工件{9}_状态"
   SymbolicIOField "符号 I/O 域_37" at 471,32 size 40x27; TextOn '1'; TextOff '0'; TextList "场次"
      ProcessValue <- "mes数据块_工件{10}_场次"
   SymbolicIOField "符号 I/O 域_38" at 471,65 size 40x27; TextOn '1'; TextOff '0'; TextList "种类"
      ProcessValue <- "mes数据块_工件{10}_种类"
   SymbolicIOField "符号 I/O 域_39" at 471,103 size 40x27; TextOn '1'; TextOff '0'; TextList "材质_1"
      ProcessValue <- "mes数据块_工件{10}_材质"
   SymbolicIOField "符号 I/O 域_40" at 471,138 size 40x27; TextOn '1'; TextOff '0'; TextList "状态_1"
      ProcessValue <- "mes数据块_工件{10}_状态"
   SymbolicIOField "符号 I/O 域_41" at 517,32 size 40x27; TextOn '1'; TextOff '0'; TextList "场次"
      ProcessValue <- "mes数据块_工件{11}_场次"
   SymbolicIOField "符号 I/O 域_42" at 517,65 size 40x27; TextOn '1'; TextOff '0'; TextList "种类"
      ProcessValue <- "mes数据块_工件{11}_种类"
   SymbolicIOField "符号 I/O 域_43" at 517,103 size 40x27; TextOn '1'; TextOff '0'; TextList "材质_1"
      ProcessValue <- "mes数据块_工件{11}_材质"
   SymbolicIOField "符号 I/O 域_44" at 517,138 size 40x27; TextOn '1'; TextOff '0'; TextList "状态_1"
      ProcessValue <- "mes数据块_工件{11}_状态"
   SymbolicIOField "符号 I/O 域_45" at 563,32 size 40x27; TextOn '1'; TextOff '0'; TextList "场次"
      ProcessValue <- "mes数据块_工件{12}_场次"
   SymbolicIOField "符号 I/O 域_46" at 563,65 size 40x27; TextOn '1'; TextOff '0'; TextList "种类"
      ProcessValue <- "mes数据块_工件{12}_种类"
   SymbolicIOField "符号 I/O 域_47" at 563,103 size 40x27; TextOn '1'; TextOff '0'; TextList "材质_1"
      ProcessValue <- "mes数据块_工件{12}_材质"
   SymbolicIOField "符号 I/O 域_48" at 563,138 size 40x27; TextOn '1'; TextOff '0'; TextList "状态_1"
      ProcessValue <- "mes数据块_工件{12}_状态"
   SymbolicIOField "符号 I/O 域_49" at 609,32 size 40x27; TextOn '1'; TextOff '0'; TextList "场次"
      ProcessValue <- "mes数据块_工件{13}_场次"
   SymbolicIOField "符号 I/O 域_50" at 609,65 size 40x27; TextOn '1'; TextOff '0'; TextList "种类"
      ProcessValue <- "mes数据块_工件{13}_种类"
   SymbolicIOField "符号 I/O 域_51" at 609,103 size 40x27; TextOn '1'; TextOff '0'; TextList "材质_1"
      ProcessValue <- "mes数据块_工件{13}_材质"
   SymbolicIOField "符号 I/O 域_52" at 609,138 size 40x27; TextOn '1'; TextOff '0'; TextList "状态_1"
      ProcessValue <- "mes数据块_工件{13}_状态"
   SymbolicIOField "符号 I/O 域_53" at 655,32 size 40x27; TextOn '1'; TextOff '0'; TextList "场次"
      ProcessValue <- "mes数据块_工件{14}_场次"
   SymbolicIOField "符号 I/O 域_54" at 655,65 size 40x27; TextOn '1'; TextOff '0'; TextList "种类"
      ProcessValue <- "mes数据块_工件{14}_种类"
   SymbolicIOField "符号 I/O 域_55" at 655,103 size 40x27; TextOn '1'; TextOff '0'; TextList "材质_1"
      ProcessValue <- "mes数据块_工件{14}_材质"
   SymbolicIOField "符号 I/O 域_56" at 655,138 size 40x27; TextOn '1'; TextOff '0'; TextList "状态_1"
      ProcessValue <- "mes数据块_工件{14}_状态"
   SymbolicIOField "符号 I/O 域_57" at 701,32 size 40x27; TextOn '1'; TextOff '0'; TextList "场次"
      ProcessValue <- "mes数据块_工件{15}_场次"
   SymbolicIOField "符号 I/O 域_58" at 701,65 size 40x27; TextOn '1'; TextOff '0'; TextList "种类"
      ProcessValue <- "mes数据块_工件{15}_种类"
   SymbolicIOField "符号 I/O 域_59" at 701,103 size 40x27; TextOn '1'; TextOff '0'; TextList "材质_1"
      ProcessValue <- "mes数据块_工件{15}_材质"
   SymbolicIOField "符号 I/O 域_60" at 701,138 size 40x27; TextOn '1'; TextOff '0'; TextList "状态_1"
      ProcessValue <- "mes数据块_工件{15}_状态"
   TextField "文本域_7" at 71,8 size 12x16; Text '1'
   TextField "文本域_8" at 117,8 size 12x16; Text '2'
   TextField "文本域_9" at 163,8 size 12x16; Text '3'
   TextField "文本域_10" at 209,8 size 12x16; Text '4'
   TextField "文本域_11" at 255,8 size 12x16; Text '5'
   TextField "文本域_12" at 301,8 size 12x16; Text '6'
   TextField "文本域_13" at 347,8 size 12x16; Text '7'
   TextField "文本域_14" at 393,8 size 12x16; Text '8'
   TextField "文本域_15" at 439,8 size 12x16; Text '9'
   TextField "文本域_16" at 485,8 size 19x16; Text '10'
   TextField "文本域_17" at 531,8 size 19x16; Text '11'
   TextField "文本域_18" at 577,8 size 19x16; Text '12'
   TextField "文本域_19" at 623,8 size 19x16; Text '13'
   TextField "文本域_20" at 669,8 size 19x16; Text '14'
   TextField "文本域_21" at 715,8 size 19x16; Text '15'
   TextField "文本域_22" at 7,178 size 44x16; Text '有无料'
   Circle "圆_1" at 63,178 size 28x28
      Appearance <- "Tag_39"
   Circle "圆_2" at 109,178 size 28x28
      Appearance <- "Tag_40"
   Circle "圆_3" at 155,178 size 28x28
      Appearance <- "Tag_41"
   Circle "圆_4" at 201,178 size 28x28
      Appearance <- "Tag_42"
   Circle "圆_5" at 247,178 size 28x28
      Appearance <- "Tag_43"
   Circle "圆_6" at 293,178 size 28x28
      Appearance <- "Tag_44"
   Circle "圆_7" at 339,178 size 28x28
      Appearance <- "Tag_45"
   Circle "圆_8" at 385,178 size 28x28
      Appearance <- "Tag_46"
   Circle "圆_9" at 431,178 size 28x28
      Appearance <- "Tag_47"
   Circle "圆_10" at 477,178 size 28x28
      Appearance <- "Tag_48"
   Circle "圆_11" at 523,178 size 28x28
      Appearance <- "Tag_49"
   Circle "圆_12" at 569,178 size 28x28
      Appearance <- "Tag_50"
   Circle "圆_13" at 615,178 size 28x28
      Appearance <- "Tag_51"
   Circle "圆_14" at 661,178 size 28x28
      Appearance <- "Tag_52"
   Circle "圆_15" at 707,178 size 28x28
      Appearance <- "Tag_53"
   TextField "文本域_23" at 16,227 size 44x16; Text '仓位号'
   TextField "文本域_24" at 23,255 size 31x16; Text '场次'
   TextField "文本域_25" at 22,288 size 31x16; Text '种类'
   TextField "文本域_26" at 22,326 size 31x16; Text '材质'
   TextField "文本域_27" at 22,361 size 31x16; Text '状态'
   SymbolicIOField "符号 I/O 域_61" at 63,251 size 40x27; TextOn '1'; TextOff '0'; TextList "场次"
      ProcessValue <- "mes数据块_工件{16}_场次"
   SymbolicIOField "符号 I/O 域_62" at 63,284 size 40x27; TextOn '1'; TextOff '0'; TextList "种类"
      ProcessValue <- "mes数据块_工件{16}_种类"
   SymbolicIOField "符号 I/O 域_63" at 63,322 size 40x27; TextOn '1'; TextOff '0'; TextList "材质_1"
      ProcessValue <- "mes数据块_工件{16}_材质"
   SymbolicIOField "符号 I/O 域_64" at 63,357 size 40x27; TextOn '1'; TextOff '0'; TextList "状态_1"
      ProcessValue <- "mes数据块_工件{16}_状态"
   SymbolicIOField "符号 I/O 域_65" at 109,251 size 40x27; TextOn '1'; TextOff '0'; TextList "场次"
      ProcessValue <- "mes数据块_工件{17}_场次"
   SymbolicIOField "符号 I/O 域_66" at 109,284 size 40x27; TextOn '1'; TextOff '0'; TextList "种类"
      ProcessValue <- "mes数据块_工件{17}_种类"
   SymbolicIOField "符号 I/O 域_67" at 109,322 size 40x27; TextOn '1'; TextOff '0'; TextList "材质_1"
      ProcessValue <- "mes数据块_工件{17}_材质"
   SymbolicIOField "符号 I/O 域_68" at 109,357 size 40x27; TextOn '1'; TextOff '0'; TextList "状态_1"
      ProcessValue <- "mes数据块_工件{17}_状态"
   SymbolicIOField "符号 I/O 域_69" at 155,251 size 40x27; TextOn '1'; TextOff '0'; TextList "场次"
      ProcessValue <- "mes数据块_工件{18}_场次"
   SymbolicIOField "符号 I/O 域_70" at 155,284 size 40x27; TextOn '1'; TextOff '0'; TextList "种类"
      ProcessValue <- "mes数据块_工件{18}_种类"
   SymbolicIOField "符号 I/O 域_71" at 155,322 size 40x27; TextOn '1'; TextOff '0'; TextList "材质_1"
      ProcessValue <- "mes数据块_工件{18}_材质"
   SymbolicIOField "符号 I/O 域_72" at 155,357 size 40x27; TextOn '1'; TextOff '0'; TextList "状态_1"
      ProcessValue <- "mes数据块_工件{18}_状态"
   SymbolicIOField "符号 I/O 域_73" at 201,251 size 40x27; TextOn '1'; TextOff '0'; TextList "场次"
      ProcessValue <- "mes数据块_工件{19}_场次"
   SymbolicIOField "符号 I/O 域_74" at 201,284 size 40x27; TextOn '1'; TextOff '0'; TextList "种类"
      ProcessValue <- "mes数据块_工件{19}_种类"
   SymbolicIOField "符号 I/O 域_75" at 201,322 size 40x27; TextOn '1'; TextOff '0'; TextList "材质_1"
      ProcessValue <- "mes数据块_工件{19}_材质"
   SymbolicIOField "符号 I/O 域_76" at 201,357 size 40x27; TextOn '1'; TextOff '0'; TextList "状态_1"
      ProcessValue <- "mes数据块_工件{19}_状态"
   SymbolicIOField "符号 I/O 域_77" at 247,251 size 40x27; TextOn '1'; TextOff '0'; TextList "场次"
      ProcessValue <- "mes数据块_工件{20}_场次"
   SymbolicIOField "符号 I/O 域_78" at 247,284 size 40x27; TextOn '1'; TextOff '0'; TextList "种类"
      ProcessValue <- "mes数据块_工件{20}_种类"
   SymbolicIOField "符号 I/O 域_79" at 247,322 size 40x27; TextOn '1'; TextOff '0'; TextList "材质_1"
      ProcessValue <- "mes数据块_工件{20}_材质"
   SymbolicIOField "符号 I/O 域_80" at 247,357 size 40x27; TextOn '1'; TextOff '0'; TextList "状态_1"
      ProcessValue <- "mes数据块_工件{20}_状态"
   SymbolicIOField "符号 I/O 域_81" at 293,251 size 40x27; TextOn '1'; TextOff '0'; TextList "场次"
      ProcessValue <- "mes数据块_工件{21}_场次"
   SymbolicIOField "符号 I/O 域_82" at 293,284 size 40x27; TextOn '1'; TextOff '0'; TextList "种类"
      ProcessValue <- "mes数据块_工件{21}_种类"
   SymbolicIOField "符号 I/O 域_83" at 293,322 size 40x27; TextOn '1'; TextOff '0'; TextList "材质_1"
      ProcessValue <- "mes数据块_工件{21}_材质"
   SymbolicIOField "符号 I/O 域_84" at 293,357 size 40x27; TextOn '1'; TextOff '0'; TextList "状态_1"
      ProcessValue <- "mes数据块_工件{21}_状态"
   SymbolicIOField "符号 I/O 域_85" at 339,251 size 40x27; TextOn '1'; TextOff '0'; TextList "场次"
      ProcessValue <- "mes数据块_工件{22}_场次"
   SymbolicIOField "符号 I/O 域_86" at 339,284 size 40x27; TextOn '1'; TextOff '0'; TextList "种类"
      ProcessValue <- "mes数据块_工件{22}_种类"
   SymbolicIOField "符号 I/O 域_87" at 339,322 size 40x27; TextOn '1'; TextOff '0'; TextList "材质_1"
      ProcessValue <- "mes数据块_工件{22}_材质"
   SymbolicIOField "符号 I/O 域_88" at 339,357 size 40x27; TextOn '1'; TextOff '0'; TextList "状态_1"
      ProcessValue <- "mes数据块_工件{22}_状态"
   SymbolicIOField "符号 I/O 域_89" at 385,251 size 40x27; TextOn '1'; TextOff '0'; TextList "场次"
      ProcessValue <- "mes数据块_工件{23}_场次"
   SymbolicIOField "符号 I/O 域_90" at 385,284 size 40x27; TextOn '1'; TextOff '0'; TextList "种类"
      ProcessValue <- "mes数据块_工件{23}_种类"
   SymbolicIOField "符号 I/O 域_91" at 385,322 size 40x27; TextOn '1'; TextOff '0'; TextList "材质_1"
      ProcessValue <- "mes数据块_工件{23}_材质"
   SymbolicIOField "符号 I/O 域_92" at 385,357 size 40x27; TextOn '1'; TextOff '0'; TextList "状态_1"
      ProcessValue <- "mes数据块_工件{23}_状态"
   SymbolicIOField "符号 I/O 域_93" at 431,251 size 40x27; TextOn '1'; TextOff '0'; TextList "场次"
      ProcessValue <- "mes数据块_工件{24}_场次"
   SymbolicIOField "符号 I/O 域_94" at 431,284 size 40x27; TextOn '1'; TextOff '0'; TextList "种类"
      ProcessValue <- "mes数据块_工件{24}_种类"
   SymbolicIOField "符号 I/O 域_95" at 431,322 size 40x27; TextOn '1'; TextOff '0'; TextList "材质_1"
      ProcessValue <- "mes数据块_工件{24}_材质"
   SymbolicIOField "符号 I/O 域_96" at 431,357 size 40x27; TextOn '1'; TextOff '0'; TextList "状态_1"
      ProcessValue <- "mes数据块_工件{24}_状态"
   SymbolicIOField "符号 I/O 域_97" at 477,251 size 40x27; TextOn '1'; TextOff '0'; TextList "场次"
      ProcessValue <- "mes数据块_工件{25}_场次"
   SymbolicIOField "符号 I/O 域_98" at 477,284 size 40x27; TextOn '1'; TextOff '0'; TextList "种类"
      ProcessValue <- "mes数据块_工件{25}_种类"
   SymbolicIOField "符号 I/O 域_99" at 477,322 size 40x27; TextOn '1'; TextOff '0'; TextList "材质_1"
      ProcessValue <- "mes数据块_工件{25}_材质"
   SymbolicIOField "符号 I/O 域_100" at 477,357 size 40x27; TextOn '1'; TextOff '0'; TextList "状态_1"
      ProcessValue <- "mes数据块_工件{25}_状态"
   SymbolicIOField "符号 I/O 域_101" at 523,251 size 40x27; TextOn '1'; TextOff '0'; TextList "场次"
      ProcessValue <- "mes数据块_工件{26}_场次"
   SymbolicIOField "符号 I/O 域_102" at 523,284 size 40x27; TextOn '1'; TextOff '0'; TextList "种类"
      ProcessValue <- "mes数据块_工件{26}_种类"
   SymbolicIOField "符号 I/O 域_103" at 523,322 size 40x27; TextOn '1'; TextOff '0'; TextList "材质_1"
      ProcessValue <- "mes数据块_工件{26}_材质"
   SymbolicIOField "符号 I/O 域_104" at 523,357 size 40x27; TextOn '1'; TextOff '0'; TextList "状态_1"
      ProcessValue <- "mes数据块_工件{26}_状态"
   SymbolicIOField "符号 I/O 域_105" at 569,251 size 40x27; TextOn '1'; TextOff '0'; TextList "场次"
      ProcessValue <- "mes数据块_工件{27}_场次"
   SymbolicIOField "符号 I/O 域_106" at 569,284 size 40x27; TextOn '1'; TextOff '0'; TextList "种类"
      ProcessValue <- "mes数据块_工件{27}_种类"
   SymbolicIOField "符号 I/O 域_107" at 569,322 size 40x27; TextOn '1'; TextOff '0'; TextList "材质_1"
      ProcessValue <- "mes数据块_工件{27}_材质"
   SymbolicIOField "符号 I/O 域_108" at 569,357 size 40x27; TextOn '1'; TextOff '0'; TextList "状态_1"
      ProcessValue <- "mes数据块_工件{27}_状态"
   SymbolicIOField "符号 I/O 域_109" at 615,251 size 40x27; TextOn '1'; TextOff '0'; TextList "场次"
      ProcessValue <- "mes数据块_工件{28}_场次"
   SymbolicIOField "符号 I/O 域_110" at 615,284 size 40x27; TextOn '1'; TextOff '0'; TextList "种类"
      ProcessValue <- "mes数据块_工件{28}_种类"
   SymbolicIOField "符号 I/O 域_111" at 615,322 size 40x27; TextOn '1'; TextOff '0'; TextList "材质_1"
      ProcessValue <- "mes数据块_工件{28}_材质"
   SymbolicIOField "符号 I/O 域_112" at 615,357 size 40x27; TextOn '1'; TextOff '0'; TextList "状态_1"
      ProcessValue <- "mes数据块_工件{28}_状态"
   SymbolicIOField "符号 I/O 域_113" at 661,251 size 40x27; TextOn '1'; TextOff '0'; TextList "场次"
      ProcessValue <- "mes数据块_工件{29}_场次"
   SymbolicIOField "符号 I/O 域_114" at 661,284 size 40x27; TextOn '1'; TextOff '0'; TextList "种类"
      ProcessValue <- "mes数据块_工件{29}_种类"
   SymbolicIOField "符号 I/O 域_115" at 661,322 size 40x27; TextOn '1'; TextOff '0'; TextList "材质_1"
      ProcessValue <- "mes数据块_工件{29}_材质"
   SymbolicIOField "符号 I/O 域_116" at 661,357 size 40x27; TextOn '1'; TextOff '0'; TextList "状态_1"
      ProcessValue <- "mes数据块_工件{29}_状态"
   SymbolicIOField "符号 I/O 域_117" at 707,251 size 40x27; TextOn '1'; TextOff '0'; TextList "场次"
      ProcessValue <- "mes数据块_工件{30}_场次"
   SymbolicIOField "符号 I/O 域_118" at 707,284 size 40x27; TextOn '1'; TextOff '0'; TextList "种类"
      ProcessValue <- "mes数据块_工件{30}_种类"
   SymbolicIOField "符号 I/O 域_119" at 707,322 size 40x27; TextOn '1'; TextOff '0'; TextList "材质_1"
      ProcessValue <- "mes数据块_工件{30}_材质"
   SymbolicIOField "符号 I/O 域_120" at 707,357 size 40x27; TextOn '1'; TextOff '0'; TextList "状态_1"
      ProcessValue <- "mes数据块_工件{30}_状态"
   TextField "文本域_28" at 77,227 size 19x16; Text '16'
   TextField "文本域_29" at 123,227 size 19x16; Text '17'
   TextField "文本域_30" at 169,227 size 19x16; Text '18'
   TextField "文本域_31" at 215,227 size 19x16; Text '19'
   TextField "文本域_32" at 261,227 size 19x16; Text '20'
   TextField "文本域_33" at 307,227 size 19x16; Text '21'
   TextField "文本域_34" at 353,227 size 19x16; Text '22'
   TextField "文本域_35" at 399,227 size 19x16; Text '23'
   TextField "文本域_36" at 445,227 size 19x16; Text '24'
   TextField "文本域_37" at 491,227 size 19x16; Text '25'
   TextField "文本域_38" at 537,227 size 19x16; Text '26'
   TextField "文本域_39" at 583,227 size 19x16; Text '27'
   TextField "文本域_40" at 629,227 size 19x16; Text '28'
   TextField "文本域_41" at 675,227 size 19x16; Text '29'
   TextField "文本域_42" at 721,227 size 19x16; Text '30'
   TextField "文本域_43" at 13,397 size 44x16; Text '有无料'
   Circle "圆_16" at 69,397 size 28x28
      Appearance <- "Tag_54"
   Circle "圆_17" at 115,397 size 28x28
      Appearance <- "Tag_55"
   Circle "圆_18" at 161,397 size 28x28
      Appearance <- "Tag_56"
   Circle "圆_19" at 207,397 size 28x28
      Appearance <- "Tag_57"
   Circle "圆_20" at 253,397 size 28x28
      Appearance <- "Tag_58"
   Circle "圆_21" at 299,397 size 28x28
      Appearance <- "Tag_59"
   Circle "圆_22" at 345,397 size 28x28
      Appearance <- "Tag_60"
   Circle "圆_23" at 391,397 size 28x28
      Appearance <- "Tag_61"
   Circle "圆_24" at 437,397 size 28x28
      Appearance <- "Tag_62"
   Circle "圆_25" at 483,397 size 28x28
      Appearance <- "Tag_63"
   Circle "圆_26" at 529,397 size 28x28
      Appearance <- "Tag_64"
   Circle "圆_27" at 575,397 size 28x28
      Appearance <- "Tag_65"
   Circle "圆_28" at 621,397 size 28x28
      Appearance <- "Tag_66"
   Circle "圆_29" at 667,397 size 28x28
      Appearance <- "Tag_67"
   Circle "圆_30" at 713,397 size 28x28
      Appearance <- "Tag_68"
   Button "按钮_1" at 10,442 size 98x32; TextOff '主画面'
      on Click: ActivateScreen("主画面", 0)
*)